// TwinCAT 3 PLC project XtsTransport
// Title: XTS Transport
// Author: D.Hauer
// ProjectVersion: 0.0.1
// Description: basic functionblocks for building XTS transport
// ProgramVersion: 3.1.4026.14
// libraries:
//   Tc2_Math, * (Beckhoff Automation GmbH)
//   Tc2_MC2, * (Beckhoff Automation GmbH)
//   Tc2_Standard, * (Beckhoff Automation GmbH)
//   Tc2_System, * (Beckhoff Automation GmbH)
//   Tc2_Utilities, * (Beckhoff Automation GmbH)
//   Tc3_McCollisionAvoidance, * (Beckhoff Automation GmbH)
//   Tc3_McCoordinatedMotion, * (Beckhoff Automation GmbH)
//   Tc3_Module, * (Beckhoff Automation GmbH)
//   Tc3_XTS_Utility, * (Beckhoff Automation GmbH)
//   VisuDialogs, * (System)
// project tree:
//   APPLICATION/ MAIN_APP.TcPOU, fb_Application.TcPOU, GVL_APPLICATION.TcGVL, PROCESS_HANDSHAKE.TcPOU
//   APPLICATION/Process_Instances/ fb_BufferInfeed.TcPOU, fb_BufferOutfeedRobot.TcPOU, fb_Infeed.TcPOU, fb_OutfeedRobot.TcPOU, fb_SenderBufferInfeed.TcPOU, fb_SenderFast.TcPOU
//   APPLICATION/_types/Application/ E_APP_CHECK.TcDUT (not stored), ST_APP_CTRL.TcDUT (not stored), ST_APP_STATE.TcDUT
//   APPLICATION/_types/Collector/ E_PROCESS_CHECK.TcDUT, E_PROCESS_CTRL.TcDUT, E_PROCESS_STATE.TcDUT (not stored), fb_ProcessCollector.TcPOU, fb_StationCollector.TcPOU, I_ProcessCollector.TcIO, ST_PROCESS_CTRL.TcDUT, ST_PROCESS_STATE.TcDUT, T_PROCESS.TcDUT
//   APPLICATION/_types/Instance/ E_INSTANCE.TcDUT, E_INSTANCE_CHECK.TcDUT (not stored), E_INSTANCE_CMD.TcDUT, E_INSTANCE_STATE.TcDUT, fb_Instance.TcPOU, ST_INSTANCE_CTRL.TcDUT (not stored), ST_INSTANCE_STATE.TcDUT
//   APPLICATION/_types/LinkedList/ fb_Process_LinkedListCtrl.TcPOU, I_Process_LinkedList.TcIO (not stored), ST_PROCESS_DATA.TcDUT, ST_PROCESS_LIST_RESULT.TcDUT (not stored)
//   APPLICATION/_Visu/ SIM_TEST.TcVIS
//   APPLICATION/_Visu/textlists/ TL_E_INSTANCE.TcTLO, TL_E_INSTANCE_CMD.TcTLO (not stored)
//   / GlobalTextList.TcGTLO, MAIN.TcPOU, PLC_1.TcTTO (not stored)
//   MSG/ fb_LocalTime.TcPOU (not stored), f_MessageSet.TcPOU (not stored), GVL_MSG.TcGVL (not stored), MessageData.TcPOU, T_MESSAGE_LIST.TcVIS
//   MSG/types/ e_Device.TcDUT (not stored), E_MessageType.TcDUT (not stored), E_MESSAGE_STATE.TcDUT, e_Subdevice.TcDUT, ST_Message.TcDUT (not stored), TL_E_MESSAGETYPE.TcTLO (not stored)
//   UML/ CD_APPLICATION.TcCD (not stored), CD_GroupCa.TcCD (not stored)
//   XTS/CaGroup/ FB_CaGroup.TcPOU, I_XtsTransport_CaGroup.TcIO
//   XTS/CaGroup/types/ E_CA_GROUP_STATE.TcDUT (not stored), E_GROUP_CHECK.TcDUT (not stored), ST_GROUP_INFO.TcDUT (not stored)
//   XTS/ GVL_XTS.TcGVL, XTS_Parameter.TcGVL
//   XTS/Mover/ fb_Mover.TcPOU, fb_MoverCtrl.TcPOU (not stored), I_XtsTransport_Mover.TcIO
//   XTS/Mover/types/ E_MOVER_CTRL.TcDUT (not stored), E_MOVER_STATE.TcDUT (not stored), ST_GEAR_DATA.TcDUT (not stored), ST_MOVER_CTRL.TcDUT (not stored), ST_MOVER_INFO.TcDUT (not stored), ST_MOVER_STATE.TcDUT (not stored), ST_MOVE_DATA.TcDUT (not stored)
//   XTS/XtsStation/ fb_Station.TcPOU, I_XtsTransport_Station.TcIO
//   XTS/XtsStation/_types/ E_STATION_CTRL.TcDUT, E_STATION_STATE.TcDUT (not stored), fb_Station_LinkedListCtrl.TcPOU, I_Station_LinkedList.TcIO (not stored), ST_STATION_CTRL.TcDUT (not stored), ST_STATION_LIST_RESULT.TcDUT (not stored), ST_STATION_MOVER_DATA.TcDUT (not stored), ST_STATION_PARAMETER.TcDUT (not stored), ST_STATION_STATE.TcDUT, T_NEST_OFFSET.TcDUT (not stored)
//   XTS/_Visualization/ GROUP_VISU.TcVIS, MOVER_VISU.TcVIS, STATION_VISU.TcVIS, Visualization Manager.TcVMO (not stored), XTS_TRANSPORT.TcVIS, XPU_VISU.TcVIS
//   XTS/_Visualization/textlists/ TL_E_CTRL_MOVER.TcTLO (not stored), TL_E_CTRL_STATION.TcTLO (not stored), TL_E_CTRL_TRANSPORT.TcTLO, TL_E_CTRL_XPU.TcTLO
//   XTS/Xpu/ fb_Xpu.TcPOU, fb_XpuCtrl.TcPOU (not stored)
//   XTS/Xpu/types/ E_XPU_CHECK.TcDUT (not stored), E_XPU_CTRL.TcDUT (not stored), E_XPU_INIT.TcDUT, E_XPU_STATE.TcDUT (not stored), ST_XPU_CTRL.TcDUT (not stored), ST_XPU_INFO.TcDUT (not stored), ST_XPU_STATE.TcDUT (not stored)
//   XTS/XtsTransportUnit/ fb_TransportUnit.TcPOU
//   XTS/XtsTransportUnit/types/ E_XTS_TRANSPORT_CHECK.TcDUT (not stored), E_XTS_TRANSPORT_CTRL.TcDUT, E_XTS_TRANSPORT_STATE.TcDUT, ST_XTS_TRANSPORT_CTRL.TcDUT (not stored), ST_XTS_TRANSPORT_STATE.TcDUT (not stored)
//   XTS/_types/ E_PROGRESS.TcDUT (not stored), f_GetProgress.TcPOU (not stored), f_GetState.TcPOU (not stored)

// ---- APPLICATION/_types/Application/ST_APP_STATE.TcDUT
TYPE ST_APP_STATE :
STRUCT
  AppState            : E_INSTANCE_STATE;
  InstanceStates      : REFERENCE TO ARRAY[1..MAX_PROCESS] OF ST_INSTANCE_STATE;
  XtsTransportState   : REFERENCE TO ST_XTS_TRANSPORT_STATE;
END_STRUCT
END_TYPE

// ---- APPLICATION/_types/Collector/E_PROCESS_CHECK.TcDUT
{attribute 'strict'}
{attribute 'to_string'}
TYPE E_PROCESS_CHECK :
(
  PROCESS_CHECK_NULL,
  PROCESS_CHECK_CTRL_REFERENCE_INVALID,
  PROCESS_CHECK_STATE_REFERENCE_INVALID,
  PROCESS_CHECK_MOVER_INFO_REFERENCE_INVALID,
	PROCESS_CHECK_STATION_FIRST_ZERO,
  PROCESS_CHECK_STATION_LAST_ZERO,
  PROCESS_CHECK_STATION_FIRST_MAX,
  PROCESS_CHECK_STATION_LAST_MAX,
  PROCESS_CHECK_STATION_COUNT_NEGATIVE, // last station must have higher index than first station, range must also be closed
  PROCESS_CHECK_STATION_COUNT_TOO_HIGH, // process can only be max (SIZEOF(T_PROCESS)*8)


  PROCESS_CHECK_DONE    := 10000
);
END_TYPE

// ---- APPLICATION/_types/Collector/E_PROCESS_CTRL.TcDUT
{attribute 'qualified_only'}
{attribute 'strict'}
{attribute 'to_string'}
TYPE E_PROCESS_CTRL :
(
  PROCESS_INIT              := 10,
  PROCESS_DISABLE           := 20,
  PROCESS_ENABLE            := 30,
  PROCESS_STATIONS_INFEED,

  PROCESS_STATIONS_ENTER    := 40,
  PROCESS_STATIONS_SEND,

  PROCESS_START             := 60,
  PROCESS_DONE              := 70,
  PROCESS_STATIONS_OUTFEED  := 80
);
END_TYPE

// ---- APPLICATION/_types/Collector/ST_PROCESS_CTRL.TcDUT
TYPE ST_PROCESS_CTRL :
STRUCT
  Cmd               : E_PROCESS_CTRL;
  ProcessTarget     : UINT;
  ActivateStation   : T_PROCESS;  // every bit is a XtsStation
  NestMask          : BYTE;       // every bit is a PosStop in a XtsStation, one mask for all XtsStations, copied to every XtsStation control in process
END_STRUCT
END_TYPE

// ---- APPLICATION/_types/Collector/ST_PROCESS_STATE.TcDUT
TYPE ST_PROCESS_STATE :
STRUCT
  State           : E_PROCESS_STATE;
  Result          : E_PROGRESS;
  Check           : E_PROCESS_CHECK;
END_STRUCT
END_TYPE

// ---- APPLICATION/_types/Collector/T_PROCESS.TcDUT
TYPE T_PROCESS : DWORD; END_TYPE

// ---- APPLICATION/_types/Instance/E_INSTANCE.TcDUT
{attribute 'qualified_only'}
//{attribute 'strict'}
{attribute 'to_string'}
TYPE E_INSTANCE :
(
  // process identifiers as enum, 
  // this enum must not have gaps!
  INVALID,
  BUFFER_INFEED,        // process for getting the job from transfersystem
  INFEED,               // process for getting workpieces from transfersystem
  //OUTFEED_CLAMP,        // process for unloading (12 movers with possible gaps)
  BUFFER_OUTFEED_ROBOT, // process for dealing movers into robot outfeed with no gaps
  OUTFEED_ROBOT_R1,     // process for robot outfeed (12 movers)
  OUTFEED_ROBOT_R2,     // process for robot outfeed (12 movers)
  //SENDER_SLOW,          // process for slowing down movers
  SENDER_FAST,          // process for accelerating movers to return with max velo
  SENDER_BUFFER_INFEED, // process for dealing movers into BUFFER_INFEED, since the curve is vertical, there has to be room when movers are set in motion
  INSTANCE_MAX
)UINT;
END_TYPE

// ---- APPLICATION/_types/Instance/E_INSTANCE_CMD.TcDUT
{attribute 'qualified_only'}
{attribute 'strict'}
{attribute 'to_string'}
TYPE E_INSTANCE_CMD : // instructions for fb_Instance executions
(
	NULL,
  INIT,
  DISABLE,
  ENABLE,
  WORK,
  PROCEED := 100,
  FINISH,
  CLEAR
)UINT;
END_TYPE

// ---- APPLICATION/_types/Instance/E_INSTANCE_STATE.TcDUT
{attribute 'qualified_only'}
//{attribute 'strict'}
{attribute 'to_string'}
TYPE E_INSTANCE_STATE :
(
  NULL,
	INVALID,
  INIT,
  DISABLED,
  DETECT_IN_LIST,
  ENABLED,
  WORKING,
  PROCEEDING,
  FINISH,
  CLEARED
)UINT;
END_TYPE

// ---- APPLICATION/_types/Instance/ST_INSTANCE_STATE.TcDUT
TYPE ST_INSTANCE_STATE :
STRUCT
  State     : E_INSTANCE_STATE;
  Progress  : E_PROGRESS;
END_STRUCT
END_TYPE

// ---- APPLICATION/_types/LinkedList/ST_PROCESS_DATA.TcDUT
TYPE ST_PROCESS_DATA :
STRUCT
  {attribute 'displaymode':='bin'}
  wTarget             : T_PROCESS; // where and how many stations are to be used in process
END_STRUCT
END_TYPE

// ---- MSG/types/E_MESSAGE_STATE.TcDUT
{attribute 'strict'}
TYPE E_MESSAGE_STATE :
(
  MSG_INVALID_POINTERS  := -1,
	MSG_NULL,
  MSG_INIT,
  MSG_ROOT              := 10,
  MSG_ROOT_CREATE,
  MSG_ROOT_CREATE_BUSY,
  MSG_FOLDER,
  MSG_FOLDER_CREATE,
  MSG_FOLDER_CREATE_BUSY,
  MSG_FILE_CREATE_DONE,
  MSG_LINE_START        := 100,
  MSG_LINE_BUILD,
  MSG_LINE_CHECK,
  MSG_WRITE_FILE_BUSY  := 200,
  MSG_WRITE_FILE_END,
  MSG_WRITE_FILE_DONE   := 1000
)DINT;
END_TYPE

// ---- MSG/types/e_Subdevice.TcDUT
{attribute 'strict'}
{attribute 'to_string'}
TYPE e_Subdevice :
(
  // sub device for message system
  General                 :=  0,
  // Motion Control FB Instances
  fbPower,
  fbReset,
  fbResetSercos,
  fbHalt,
  fbStop,                 // 5
  fbHome,
  fbJog,
  fbMoveVelocity1,
  fbMoveVelocity2,
  fbMoveAbsolute1,        // 10
  fbMoveAbsolute2,
  fbMoveEndless,
  fbMovePtP,
  fbMoveVelo,

  // CA CollisionAvoidance FB instances
  // CA group fb instances
  fbCaGroup             := 30,
  fbMoveToPosCa,
  fbSendToAbsPosCa,
  fbSendToModuloPosCa,
  fbGearInPosCa,
  fbGroupAddAxis,
  fbGroupRemoveAxis,
  fbGroupDisable,
  fbGroupEnable,
  fbGroupErrorRead,
  fbGroupStatusRead,
  fbGroupReset,
  fbGroupStop,
  fbHaltCa,

  fbGearIn                := 50,
  fbGearOut,
  fbGearInMultiMaster,

  fbCamOutV2              := 80,
  fbCamInV2,
  fbCamScalingV2,
  fbCamInfoV2,
  fbReadMotionFunction,
  fbReadMotionFunctionPoint,
  fbReadMotionFunctionValues,
  fbWriteMotionFunction,
  fbWriteMotionFunctionPoint,
  fbSetOnlineChangeMode,

  fbReadParameter         := 100,
  fbReadBoolParameter,
  fbWriteParameter,
  fbWriteBoolParameter,
  fbWriteParameterPersistent,

  fbBuildGroup            := 200,
  fbClearGroup,
  fbLoadProg,
  fbResetItp,
  fbStartStopItp,
  fbEStopItp,             // 205
  fbStepOnAfterEStopItp,
  fbConfirmHskItp,
  fbDelDtgItp,
  fbNciFeedTablePreparation,
  fbNciFeedTable,         // 210
  fbReadLine,
  fbItpReadRParams,
  fbItpWriteRParams,
  Get_ItpState,
  Get_Error,              // 215


  XfcPositionAtTime       := 300,
  XfcTimeOfPosition,
  XfcTimeToPosition,
  XfcTimeToModuloPosition,
  XfcRecordedPosition,
  XfcTouchProbe,          // 305
  XfcTouchProbeEL1258,
  XfcTouchProbeOptions,
  XfcTriggerRef,
  XfcTriggerRef_MT,
  XfcEl1258Interface_MT,  // 310
  XfcRecordedPosition_MT,
  XfcTriggerOut,
  XfcTriggerStart,
  XfcSwitchOn_2252,
  XfcSwitchOff_2252,      // 315
  XfcInit,
  XfcLatchPosition,
  XfcWaitForPosition,

  AxisMode              := 1000,
  AxisControl,

  NciControl            := 2000,
  NciStartUp,
  NciCycle,
  NciIdle,

  StationLinkedList     := 3000,
  StationInitList,
  StationAddHead,
  StationAddTail,
  StationGetHead,
  StationRemoveHeadValue,

  StationControl        := 4000,
  StationState, 

  Xpu_fbEnvironment     := 5000,
  Xpu_fbProcessingUnit,
  Xpu_fbXpuPart,
  Xpu_fbXpuTrack,
  Xpu_fbMc2CaGroup,
  Xpu_fbParameterSet,

  Xpu_fbPartModules     := 5500,

  Xpu_fbMoverXpu        := 6000,

  TransportUnit_General := 7000,
  TransportUnit_Restart := 7010,
  TransportUnit_Start,
  TransportUnit_XpuInit,

  CamControl            := 8000,
  CamStartUp,
  CamCycle,

  Process_StationCollector    := 11000,
  Process_ProcessCollector    := 11100,
  Process_ProcessCollector_Init,
  Process_ProcessCollector_Cycle,
  Process_ProcessCollector_Control,

  Process_LinkedList_GetHead,
  Process_LinkedList_RemoveHead,
  Process_LinkedList_AddTail,
  Process_LinkedList_CheckData,

  Instance_BufferInfeed       := 12000,
  Instance_BufferInfeed_CheckDisabled,
  Instance_BufferInfeed_CheckEnabled,
  Instance_BufferInfeed_CheckInfeed,
  Instance_BufferInfeed_CheckOutfeed,
  Instance_BufferInfeed_CheckTarget,
  Instance_Infeed,
  Instance_BufferOutfeedRobot,
  Instance_OutfeedRobot_R1,
  Instance_OutfeedRobot_R2,
  Instance_Sender_Fast,
  Instance_Sender_BufferInfeed,

  Application                 := 13000,
  Application_Check,
  Application_Clear,
  Application_Cmd,
  Application_Disable,
  Application_Enable,
  Application_Finish,
  Application_Init,
  Application_Proceed,
  Application_Work

)DINT;
END_TYPE

// ---- XTS/XtsStation/_types/E_STATION_CTRL.TcDUT
{attribute 'qualified_only'}
{attribute 'strict'}
{attribute 'to_string'}
TYPE E_STATION_CTRL :
(
  STATION_CTRL_NULL,              // nothing happens here
	STATION_INIT            := 1,   // hard reset of station, list is cleared
  STATION_DISABLE         := 10,  // 
  STATION_ENABLE,                 // 

  STATION_MOVER_ENTER     := 20,  // mover may enter station
  STATION_MOVER_ENTER_RETRY,      // retry after E_STATION_STATE.STATION_ERROR_INFEED_ERROR
  STATION_MOVER_SEND,             // do not enter, send to E_STATION_STATE.STATION_MOVER_OUT

  STATION_PROCESS_START   := 30,  // double handshake with extern
  STATION_PROCESS_DONE,           // single handshake with extern

  STATION_MOVER_OUT       := 50,  // mover may leave station now; ticket for mover is checked here (ST_STATION_CTRL.nTargetStation)
  STATION_MOVER_OUT_RETRY,        // retry after E_STATION_STATE.STATION_ERROR_OUTFEED_ERROR

  STATION_MOVER_GONE      := 60   // mover has left station, last handshake station is empty

)USINT;
END_TYPE

// ---- XTS/XtsStation/_types/ST_STATION_STATE.TcDUT
{attribute 'pack_mode' := '2'}
TYPE ST_STATION_STATE :
STRUCT
  eState          : E_STATION_STATE;
  {attribute 'displaymode':='bin'}
  nMask           : BYTE;
  nMoverId        : USINT;
  rMoverModPos    : LREAL; // modulo position of detected mover
  rMoverVelo      : LREAL;
  rMoverAcc       : LREAL;
  nQueue          : USINT; // queue count for station
END_STRUCT
END_TYPE

// ---- XTS/Xpu/types/E_XPU_INIT.TcDUT
{attribute 'to_string'}
TYPE E_XPU_INIT :
(
	INIT_START,
  INIT_ENVIRONMENT_OID            := 10,
  INIT_INFO_SERVER_ITF,
  INIT_INFO_SERVER_STATION_COUNT,
  INIT_INFO_SERVER_STATION_OID,
  INIT_CA_GROUP_OID               := 20,
  INIT_CA_GROUP_GET_OID,
  INIT_CA_GROUP_CHECK_OID,
  INIT_CA_GROUP_COM,
  INIT_PARAMETERSET_COUNT,
  INIT_PARAMETERSET_OID,
  INIT_PARAMETERSET_COM,
  INIT_PARAMETERSET_COM_NEXT,
  INIT_PROCESSING_UNIT_COM        := 30,
  INIT_PROCESSING_UNIT_PART_COUNT,
  INIT_PROCESSING_UNIT_PART_OID,
  INIT_PROCESSING_UNIT_TRACK_COUNT,
  INIT_PROCESSING_UNIT_TRACK_OID,
  INIT_PROCESSING_UNIT_MOVER_COUNT,
  INIT_PROCESSING_UNIT_MOVER_OID,
  INIT_PROCESSING_UNIT_TASK_COUNT,
  INIT_PROCESSING_UNIT_TASK_OID,
  INIT_TRACK_COM                  := 50,
  INIT_PART_COM                   := 60,
  INIT_PART_MODULE_COUNT,
  INIT_PART_MODULE_OID,
  INIT_PART_MODULE_COM,
  INIT_PART_MODULE_COM_NEXT,
  INIT_MOVER_COM                  := 70,
  INIT_MOVER_COM_NEXT,
  INIT_DATA_GET                   := 90,
  INIT_DATA_CHECK,
  INIT_DONE                       := 100
)UINT;
END_TYPE

// ---- XTS/XtsTransportUnit/types/E_XTS_TRANSPORT_CTRL.TcDUT
{attribute 'strict'}
{attribute 'to_string'}
TYPE E_XTS_TRANSPORT_CTRL :
(
  CMD_NULL,
  CMD_INIT                  := 10,  // Xpu, Group, Mover initialization: clear errors, clear group, check Xpu data, check mover detection
  CMD_IDLE,

  CMD_MOVER_ENABLE          := 20,  // all mover are enabled, checked for ControlLoopClosed
  CMD_MOVER_DISABLE,                // all mover are disabled, no axis in CaGroup: no error, any axis in CaGroup: group error
  CMD_MOVER_HALT_CA,                // all movers are stopped with MC_HaltCA[]. ONLY use if all movers are in CA group

  CMD_GROUP_CLEAR           := 30,  // halt all movers, clear errors, remove all movers from group, clear group
  CMD_GROUP_BUILD,                  // add all movers to group
  CMD_GROUP_ENABLE,                 // group with movers is enabled
  CMD_GROUP_STOP,                   // moving CA Group is stopped

  CMD_TRANSPORT_START       := 40,  // move all mover[i] to start position
  CMD_TRANSPORT_RESTART             // move all mover[i] to LastPosition[i]

)UINT;
END_TYPE

// ---- XTS/XtsTransportUnit/types/E_XTS_TRANSPORT_STATE.TcDUT
{attribute 'to_string'}
TYPE E_XTS_TRANSPORT_STATE :
(
  TRANSPORT_NULL,
  TRANSPORT_INVALID,
  TRANSPORT_INIT            := 10,  // Xpu, Group, Mover initialization: init TcCOM objects, clear errors, clear group, check Xpu data, check mover detection
  TRANSPORT_IDLE,                   // cyclic check for errors, check Xpu data

  TRANSPORT_MOVER_ENABLE    := 20,  // all mover are enabled, checked for ControlLoopClosed
  TRANSPORT_MOVER_DISABLE,          // all mover are disabled
  TRANSPORT_MOVER_HALT_CA,          // all mover standstill
  TRANSPORT_MOVER_STOP,

  TRANSPORT_GROUP_CLEAR     := 30,  // halt all movers, clear errors, remove all movers from group, clear group
  TRANSPORT_GROUP_BUILD,            // add all movers to group
  TRANSPORT_GROUP_ENABLE,           // group with movers is enabled
  TRANSPORT_GROUP_STOP,             // CaGroup Stop, CaGroup Reset, All movers halt

  TRANSPORT_START           := 40,  // move all mover[i] to start position
  TRANSPORT_RESTART                 // move all mover[i] to LastPosition[i]
)UINT;
END_TYPE

// ---- APPLICATION/GVL_APPLICATION.TcGVL
VAR_GLOBAL CONSTANT
  MAX_PROCESS         : E_INSTANCE := E_INSTANCE.SENDER_BUFFER_INFEED;
END_VAR
{attribute 'qualified_only'}
VAR_GLOBAL
  //-----------------------------------------------------------------------------------------------
  // Application
  //
  //  this is the part you will have to change and adapt into your programming
  //-----------------------------------------------------------------------------------------------
  //-----------------------------------------------------------------------------------------------
  // fb_Application:
  // - procedures for getting fb_Instance classes and XTS_TRANSPORT_LAYER to work
  //
  //  - Cmd/state behaviour as in fb_TransportUnit
  //  - E_INSTANCE_CMD  / E_INSTANCE_STATE + E_PROGRESS
  //      INIT          /   INIT          : initialize processes and XtsStations       
  //      DISABLE       /   DISABLED      : RemoveAllAxis from CA Group, disable CA Group, disable all movers
  //      ENABLE        /   ENABLED       : AddAllAxis to CA Group, Enable CA Group, Enable all movers
  //      WORK          /   WORKING       : CMD_TRANSPORT_START, enable handshakes, start writing list entries to BUFFER_INFEED
  //      PROCEED       /   PROCEEDING    : CMD_TRANSPORT_RESTART, enable handshakes, continue writing list entries to BUFFER_INFEED
  //      FINISH        /   FINISH        : stop writing list entries to BUFFER_INFEED, handshake processes until outfeeds are empty
  //      CLEAR         /   CLEARED       : clear all instances of fb_Instance, clear all XtsStations
  //-----------------------------------------------------------------------------------------------
  ApplicationMain       : fb_Application;
  AppControl            : ST_APP_CTRL;
  AppState              : ST_APP_STATE;


  //-----------------------------------------------------------------------------------------------
  // Process instances
  //  - processes are similar but also different, hence working with inheritance of fb_Instance
  //  - change/check here if you need a process procedure that matches your use case
  //-----------------------------------------------------------------------------------------------
  BufferInfeed          : fb_BufferInfeed;        // prepare movers to enter infeed station
  Infeed                : fb_Infeed;              // infeed into XTS, transfersystem drops its load here
  BufferOutfeedRobot    : fb_BufferOutfeedRobot;  // feeds 24 Mover into 2 processes (12 each), no gaps
  Outfeed_R1            : fb_OutfeedRobot;        // unloads 12 mover
  Outfeed_R2            : fb_OutfeedRobot;        // unloads 12 mover
  SenderFast            : fb_SenderFast;          // every passing mover is accelersted to max velo
  SenderBufferInfeed    : fb_SenderBufferInfeed;  // checks if there is room for 12-x mover, sends mover to BufferInfeed for a new round


  //-----------------------------------------------------------------------------------------------
  // fb_Instance control and state
  //  - structs are used in fb_Application as reference 
  //-----------------------------------------------------------------------------------------------
  InstanceCtrl          : ARRAY[1..MAX_PROCESS] OF ST_INSTANCE_CTRL;
  InstanceState         : ARRAY[1..MAX_PROCESS] OF ST_INSTANCE_STATE;


  //-----------------------------------------------------------------------------------------------
  // Linked List instances
  //  - THIS example only uses the linked list in fb_BufferInfeed 
  //    as buffered input from an extern transfersystem
  //-----------------------------------------------------------------------------------------------
  ProcessList           : ARRAY[1..MAX_PROCESS] OF fb_Process_LinkedListCtrl; // information transfer between processes
  ItfProcessList        : ARRAY[1..MAX_PROCESS] OF I_Process_LinkedList;      // use this interface in your function blocks


  //-----------------------------------------------------------------------------------------------
  // Collector instances
  //
  //  - layer for grouping parallel XtsStations for process handshakes
  //-----------------------------------------------------------------------------------------------
  //  - fb_ProcessCollector:
  //    - uses .ProcessCtrl and .ProcessState for handshakes with application
  //
  //    - .ActivateStation is evaluated after enabling infeed in state 
  //      E_PROCESS_STATE.PROCESS_DISABLE:/E_PROGRESS.PROGRESS_BUSY:
  //      
  //    - ST_PROCESS_STATE:
  //      - contains 3 enumerations for you to check
  //      - State           : E_PROCESS_STATE;
  //        - main state for handshakes
  //
  //      - Result          : E_PROGRESS;
  //        - substate for checks during handshake; 
  //          PROGRESS_BUSY --> handshakes are accepted (see fb_ProcessCollecotr.Cycle())
  //
  //      - Check           : E_PROCESS_CHECK;
  //        - cyclic pointer check: use this on startup of your application
  //
  //    - inherits fb_StationCollector
  //-----------------------------------------------------------------------------------------------
  ProcessCollector      : ARRAY[1..MAX_PROCESS] OF fb_ProcessCollector;       // grouping of XtsStations
  ItfProcessCollector   : ARRAY[1..MAX_PROCESS] OF I_ProcessCollector;        // interface for use in your function blocks like BufferInfeed etc.
END_VAR

// ---- XTS/GVL_XTS.TcGVL
{attribute 'qualified_only'}
VAR_GLOBAL
  //---------------------------------------------------------------------------
  // XTS Station
  //  - handshakes mover in station with extern control
  //  - station parameters (positions, gap, dyn. constraints, description...)
  StationStart        : ST_STATION_PARAMETER;   // Xts transport is sending all mover to this position (CMD_TRANSPORT_START)
  StationStartIndex   : UINT := 52;             // index of XtsStation where all movers are entered into linked list.

  // station handshaking with mover and extern process
  // station sends mover to target station/WaitPos
  // station adds mover data to LinkedList.AddTail() of target station
  Station             : ARRAY[1..MAX_STATION] OF fb_Station;
  StationList         : ARRAY[1..MAX_STATION] OF fb_Station_LinkedListCtrl;

  StationQueue        : ARRAY[1..MAX_STATION]    OF 
                        ARRAY[1..MAX_LIST_NODES] OF ST_STATION_MOVER_DATA;

  // interface for access to List methods
  StationListItf      : ARRAY[1..MAX_STATION] OF I_Station_LinkedList;

  // interface for access to station methods
  StationCtrlItf      : ARRAY[1..MAX_STATION] OF I_XtsTransport_Station;

  // ctrl / state datafields for extern control
  StationCtrl         : ARRAY[1..MAX_STATION] OF ST_STATION_CTRL;   // control for extern to write
  StationState        : ARRAY[1..MAX_STATION] OF ST_STATION_STATE;  // state for extern to read

  // station parameter
  StationParameter    : ARRAY[1..MAX_STATION] OF ST_STATION_PARAMETER;

  // static position offsets in stations
  PositionOffset      : ARRAY[1..MAX_STATION] OF T_NEST_OFFSET;


  //---------------------------------------------------------------------------
  // XTS
  // XTS TransportUnit
  //  - handles request for XPU, Group, Mover, StartUp, ReStart
  XtsTransport        : fb_TransportUnit;         // manages members of XTS transport for extern to access

  XtsTransportCtrl    : ST_XTS_TRANSPORT_CTRL;    // control of XTS transport for extern to write
  XtsTransportState   : ST_XTS_TRANSPORT_STATE;   // state   of XTS transport for extern to read


  //---------------------------------------------------------------------------
  // XPU
  // XTS-Utility checks
  Xpu             : fb_XpuCtrl;

  XpuCtrl         : ST_XPU_CTRL;
  XpuState        : ST_XPU_STATE;
  XpuInfo         : ST_XPU_INFO;
  XpuModules      : ARRAY[1..MAX_MODULE] OF Tc3_XTS_Utility.ST_InfoDataView;


  //---------------------------------------------------------------------------
  // Collision avoidance group CA
  //
  // - add mover to group
  // - build group
  // - clear group
  CaGroup         : FB_CaGroup;                   // cyclic check of CaGroup state and errors; carries methods for handling CaGroup
  CaGroupItf      : I_XtsTransport_CaGroup;       // Interface used by fb_TransportUnit

  // cyclic mapping to MOTION/Objects/CaGroup 
  CaGroupRef      : Tc3_McCoordinatedMotion.AXES_GROUP_REF;

  // Info data from CaGroup FB
  CaGroupInfo     : ST_GROUP_INFO;                // cyclic info about CaGroup for fb_TransportUnit to read
  //---------------------------------------------------------------------------

  //---------------------------------------------------------------------------
  // MC2 encapsulation, CA movement
  Mover           : ARRAY[1..MAX_MOVER] OF fb_MoverCtrl;    // MC and CA methods for mover; cyclic check for individual command on mover

  MoverCtrl       : ARRAY[1..MAX_MOVER] OF ST_MOVER_CTRL;   // control of individual mover for extern to write
  MoverState      : ARRAY[1..MAX_MOVER] OF ST_MOVER_STATE;  // state   of individual mover for extern to read

  MoverItf        : ARRAY[1..MAX_MOVER] OF I_XtsTransport_Mover;  // Interface used by fb_TransportUnit

  LastPosition    : ARRAY[1..MAX_MOVER] OF LREAL;           // on execute of any movement, value is saved here (used by fb_Mover)
  LastGap         : ARRAY[1..MAX_MOVER] OF LREAL;           // on execute of any movement, value is saved here (used by fb_Mover)

  MoverInfo       : ARRAY[1..MAX_MOVER] OF ST_MOVER_INFO;   // cyclic info about mover for extern to read

  MoveData        : ARRAY[1..MAX_MOVER] OF ST_MOVE_DATA;    // dynamic constraints for move commands
  GearData        : ARRAY[1..MAX_MOVER] OF ST_GEAR_DATA;    // dynamic constraints and positions for GearIn/GearInPosCa
  
  // cyclic mapping to MOTION/Axes
  AxisRefMover    : ARRAY[1..MAX_MOVER] OF Tc2_MC2.AXIS_REF;
  //---------------------------------------------------------------------------
END_VAR

// ---- XTS/XTS_Parameter.TcGVL
//{attribute 'qualified_only'}
VAR_GLOBAL CONSTANT
// HAUD 2025 06 04
//
//    XTS_TRANSPORT_LAYER project
//    
//    MIT License
//    
//    Copyright (c) 2025 HAUD
//    
//    Permission is hereby granted, free of charge, to any person obtaining a copy
//    of this software and associated documentation files (the "Software"), to deal
//    in the Software without restriction, including without limitation the rights
//    to use, copy, modify, merge, publish, distribute, sublicense, and/or sell
//    copies of the Software, and to permit persons to whom the Software is
//    furnished to do so, subject to the following conditions:
//    
//    The above copyright notice and this permission notice shall be included in all
//    copies or substantial portions of the Software.
//    
//    THE SOFTWARE IS PROVIDED "AS IS", WITHOUT WARRANTY OF ANY KIND, EXPRESS OR
//    IMPLIED, INCLUDING BUT NOT LIMITED TO THE WARRANTIES OF MERCHANTABILITY,
//    FITNESS FOR A PARTICULAR PURPOSE AND NONINFRINGEMENT. IN NO EVENT SHALL THE
//    AUTHORS OR COPYRIGHT HOLDERS BE LIABLE FOR ANY CLAIM, DAMAGES OR OTHER
//    LIABILITY, WHETHER IN AN ACTION OF CONTRACT, TORT OR OTHERWISE, ARISING FROM,
//    OUT OF OR IN CONNECTION WITH THE SOFTWARE OR THE USE OR OTHER DEALINGS IN THE
//    SOFTWARE.

  Version             : STRING  := '4.00.08';

  MAX_MOVER           : UINT    := TO_UINT(Tc3_XTS_Utility.TcIoXtsEnvironmentParameterList.MaxXtsMoversPerXpu);
  MAX_MODULE          : UINT    := TO_UINT(Tc3_XTS_Utility.TcIoXtsEnvironmentParameterList.MaxModulesPerPart);
  MAX_PART            : UINT    := TO_UINT(Tc3_XTS_Utility.TcIoXtsEnvironmentParameterList.MaxXtsPartsPerXpu);
  MAX_TRACK           : UINT    := TO_UINT(Tc3_XTS_Utility.TcIoXtsEnvironmentParameterList.MaxXtsTracksPerXpu);
  MAX_GROUP           : UINT    := TO_UINT(Tc3_XTS_Utility.TcIoXtsEnvironmentParameterList.MaxXtsCaGroup);

  MAX_INFO_SERVER     : UINT    := TO_UINT(Tc3_XTS_Utility.TcIoXtsEnvironmentParameterList.MaxXtsInfoServer);
  MAX_INFO_STATION    : UINT    := TO_UINT(Tc3_XTS_Utility.TcIoXtsEnvironmentParameterList.MaxXtsInfoStation);
  MAX_INFO_STOP_POS   : UINT    := TO_UINT(Tc3_XTS_Utility.TcIoXtsEnvironmentParameterList.MaxXtsStopPositionsPerStation);

  MAX_PARAMETER_SET   : UINT    := TO_UINT(Tc3_XTS_Utility.TcIoXtsEnvironmentParameterList.MaxXtsParameterSet);

  MAX_NCT_BASE_UNIT   : UINT    := TO_UINT(Tc3_XTS_Utility.TcIoXtsEnvironmentParameterList.MaxXtsNctBaseUnitInterfaces);

  MAX_STATION         : UINT    := 53;
  MAX_STATION_NEST    : UINT    := TO_UINT(SIZEOF(ST_STATION_STATE.nMask)*8);
  // MAX_LIST_NODES      : UINT    := MAX_MOVER;
  MAX_LIST_NODES      : UINT    := 108; // visualization can not handle access to MAX_MOVER
  MAX_MASTER          : UINT    := 1;
END_VAR

// ---- APPLICATION/_types/Collector/I_ProcessCollector.TcIO
INTERFACE I_ProcessCollector

PROPERTY ActivateStation : DWORD // bit mask for enabling XtsStations in Process
GET
END_GET
END_PROPERTY

METHOD BitsToString : STRING(SIZEOF(T_PROCESS)*8) // T_PROCESS to string
VAR_INPUT
  inVal       : T_PROCESS;
END_VAR
END_METHOD

METHOD Cycle // cyclic call for checking XtsStation state masks and command input from process
END_METHOD

METHOD PUBLIC DelBit : T_PROCESS
VAR_INPUT
  inVal   : T_PROCESS;
  bitNo   : DINT;
END_VAR
END_METHOD

METHOD PUBLIC GetBit : BOOL
VAR_INPUT
  inVal   : T_PROCESS;
  bitNo   : DINT;
END_VAR
END_METHOD

METHOD GetMoverInStation : ST_MOVER_INFO // mover in station info
VAR_INPUT
  nStation            : UINT;   // index of GVL_XTS.StationState[nStation]
END_VAR
END_METHOD

METHOD GetStationState : ST_STATION_STATE
VAR_INPUT
  nStation            : UINT;   // index of GVL_XTS.StationState[nStation]
END_VAR
END_METHOD

METHOD PUBLIC Init : E_PROGRESS // clears all XtsSubstations, then disables all
VAR_INPUT
  Execute     : BOOL;
END_VAR
END_METHOD

PROPERTY MessageLevel : e_MessageType
GET
END_GET
SET
END_SET
END_PROPERTY

PROPERTY ProcessCtrl : reference to st_process_ctrl
GET
END_GET
SET
END_SET
END_PROPERTY

PROPERTY ProcessId : E_INSTANCE
GET
END_GET
SET
END_SET
END_PROPERTY

PROPERTY ProcessState : reference to st_process_state
GET
END_GET
SET
END_SET
END_PROPERTY

PROPERTY QueueMoverIDs : ARRAY[1..SIZEOF(T_PROCESS)*8] OF UINT
GET
END_GET
END_PROPERTY

PROPERTY QueueProcessCount : UINT // sum of all station queues
GET
END_GET
END_PROPERTY

PROPERTY QueueStationCount : ARRAY[1..SIZEOF(T_PROCESS)*8] OF UINT
GET
END_GET
END_PROPERTY

METHOD PUBLIC SetBit : T_PROCESS
VAR_INPUT
  inVal   : T_PROCESS;
  bitNo   : DINT;
END_VAR
END_METHOD

PROPERTY StationCount : UINT
GET
END_GET
END_PROPERTY

PROPERTY StationFirst : uint
GET
END_GET
SET
END_SET
END_PROPERTY

PROPERTY StationLast : uint
GET
END_GET
SET
END_SET
END_PROPERTY

PROPERTY TargetIndex : ARRAY[1..SIZEOF(T_PROCESS)*8] OF USINT
GET
END_GET
SET
END_SET
END_PROPERTY

PROPERTY TargetMask : ARRAY[1..SIZEOF(T_PROCESS)*8] OF BYTE
GET
END_GET
SET
END_SET
END_PROPERTY

METHOD To_T_Process : T_PROCESS // maps (2^nExp)-1 onto T_PROCESS datatype 
VAR_INPUT
  nExp              : BYTE;
END_VAR
END_METHOD

END_INTERFACE

// ---- XTS/CaGroup/I_XtsTransport_CaGroup.TcIO
INTERFACE I_XtsTransport_CaGroup

METHOD AddAll : E_PROGRESS
VAR_INPUT
  Execute     : BOOL;
END_VAR
END_METHOD

METHOD Disable : E_PROGRESS
VAR_INPUT
  Execute     : BOOL;
END_VAR
END_METHOD

METHOD Enable : E_PROGRESS
VAR_INPUT
  Execute     : BOOL;
END_VAR
END_METHOD

METHOD McHaltAll : E_PROGRESS
VAR_INPUT
  Execute       : BOOL;
END_VAR
END_METHOD

METHOD McResetAll : E_PROGRESS
VAR_INPUT
  Execute       : BOOL;
END_VAR
END_METHOD

METHOD RemoveAll : E_PROGRESS
VAR_INPUT
  Execute     : BOOL;
END_VAR
END_METHOD

METHOD Reset : E_PROGRESS
VAR_INPUT
  Execute     : BOOL;
END_VAR
END_METHOD

METHOD Stop : E_PROGRESS
VAR_INPUT
  Execute     : BOOL;
END_VAR
END_METHOD

END_INTERFACE

// ---- XTS/Mover/I_XtsTransport_Mover.TcIO
INTERFACE I_XtsTransport_Mover

METHOD Disable : E_PROGRESS
VAR_INPUT
  Execute             : BOOL;
END_VAR
END_METHOD

METHOD Enable : E_PROGRESS
VAR_INPUT
  Execute             : BOOL;
END_VAR
END_METHOD

METHOD GearIn : E_PROGRESS;
VAR_INPUT
  Execute             : BOOL;
  stMoveData          : ST_MOVE_DATA;
  stGearData          : ST_GEAR_DATA;
END_VAR
END_METHOD

METHOD GearInPosCa : E_PROGRESS
VAR_INPUT
  Execute             : BOOL;
  stMoveData          : ST_MOVE_DATA;
  stGearData          : ST_GEAR_DATA;  
END_VAR
END_METHOD

METHOD GearOut : E_PROGRESS
VAR_INPUT
  Execute             : BOOL;
END_VAR
END_METHOD

METHOD Halt : E_PROGRESS
VAR_INPUT
  Execute             : BOOL;
  stMoveData          : ST_MOVE_DATA;
END_VAR
END_METHOD

METHOD HaltCa : E_PROGRESS
VAR_INPUT
  Execute             : BOOL;
  stMoveData          : ST_MOVE_DATA;
END_VAR
END_METHOD

PROPERTY MessageLevel : e_messagetype
SET
END_SET
END_PROPERTY

PROPERTY ModuloTurn : dint
GET
END_GET
END_PROPERTY

METHOD MoveToPos : E_PROGRESS
VAR_INPUT
  Execute             : BOOL;
  stMoveData          : ST_MOVE_DATA;
END_VAR
END_METHOD

METHOD MoveToPosCa : E_PROGRESS
VAR_INPUT
  Execute             : BOOL;
  stMoveData          : ST_MOVE_DATA;
END_VAR
END_METHOD

PROPERTY RailLength : LREAL
GET
END_GET
SET
END_SET
END_PROPERTY

METHOD Reset : E_PROGRESS
VAR_INPUT
  Execute             : BOOL;
END_VAR
END_METHOD

METHOD SendToAbsPosCa : E_PROGRESS
VAR_INPUT
  Execute             : BOOL;
  stMoveData          : ST_MOVE_DATA;
END_VAR
END_METHOD

METHOD SendToModuloPosCa : E_PROGRESS
VAR_INPUT
  Execute             : BOOL;
  stMoveData          : ST_MOVE_DATA;
END_VAR
END_METHOD

END_INTERFACE

// ---- XTS/XtsStation/I_XtsTransport_Station.TcIO
INTERFACE I_XtsTransport_Station

METHOD Init : e_progress
VAR_INPUT
END_VAR
END_METHOD

END_INTERFACE

// ---- APPLICATION/fb_Application.TcPOU
//---------------------------------------------------------------------------------------------------------------
//
//  HAUD 2025.03.31
//
//  - EXAMPLE for top level procedures
//    - transport layer
//    - Collector layer
//    - process layer
//    - instance ctrl/state
//
//  - rewrite/change/discard as you require for your application
//
//  - this function block is NOT intended for direct use outside the scope of this example
//  - maybe the command mechanics are useful for your application
//
//---------------------------------------------------------------------------------------------------------------
FUNCTION_BLOCK fb_Application
VAR
  _eCheck                       : E_APP_CHECK;
  _eInit                        : E_PROGRESS;

  _Ctrl                         : REFERENCE TO ST_APP_CTRL;
  _State                        : REFERENCE TO ST_APP_STATE;

  _eResult                      : E_PROGRESS;

  _eCmd,
  _eCmdOld                      : E_INSTANCE_CMD;
  _eState                       : E_INSTANCE_STATE;

  // Transport Ctrl/State
  _XtsTransportCtrl             : REFERENCE TO ST_XTS_TRANSPORT_CTRL;
  _XtsTransportState            : REFERENCE TO ST_XTS_TRANSPORT_STATE;

  _InstanceCtrl                 : REFERENCE TO ARRAY[1..MAX_PROCESS] OF ST_INSTANCE_CTRL;
  _InstanceState                : REFERENCE TO ARRAY[1..MAX_PROCESS] OF ST_INSTANCE_STATE;
  
  _ItfProcessCollector          : REFERENCE TO ARRAY[1..MAX_PROCESS] OF I_ProcessCollector;

  _ItfProcessList               : REFERENCE TO ARRAY[1..MAX_PROCESS] OF I_Process_LinkedList;

  // timers for this example
  _tonProcess                   : ARRAY[1..MAX_PROCESS] OF Tc2_Standard.TON;
  _tProcess                     : ARRAY[1..MAX_PROCESS] OF TIME;


  _stMsg                        : ST_Message;
  _MessageLevel                 : E_MessageType;

  // ListData()
  _nLoadCaseOld,
  _nLoadCase                    : UINT := 0; // 0 = fully loaded, 2 = mod 5 missing 1, 1 = missing up to 11

  // Work()
  _bSingleOutput                : BOOL;

  _nTimeVariantOld,
  _nTimeVariant                 : UINT;

  _sAppState                    : STRING;
  _sAppResult                   : STRING;

  {attribute 'hide'}
  _nAppState                    : E_INSTANCE_STATE;
  {attribute 'hide'}
  _nAppResult                   : E_PROGRESS;
END_VAR

IF NOT Check() THEN RETURN; END_IF
//-----------------------------------------------------------------------------
//-----------------------------------------------------------------------------
// set message device
//-----------------------------------------------------------------------------
_stMsg.eDevice                  := e_Device.Application + 1;

_eCmd                           := _Ctrl.Cmd;
// check for command change
// get state for cmd
IF (_eCmd <> _eCmdOld)
THEN
  _eState                       := Cmd(_eCmd);
  _eCmdOld                      := _eCmd;

  IF (_MessageLevel > E_MessageType.eMessageWarning)
  THEN
    _stMsg.eType                      := E_MessageType.eMessageinfo;
    _stMsg.eSubdevice                 := e_Subdevice.Application_Cmd;
    _stMsg.iErrorNumber               := _eCmd;
    _stMsg.sText                      := concat(TO_STRING(_eCmd), ': ');
    _stMsg.sText                      := concat(_stMsg.sText, TO_STRING(_eState));
    f_MessageSet(_stMsg);
  END_IF
END_IF

CASE _eResult
OF
  E_PROGRESS.PROGRESS_INVALID:
    _State.AppState             := TO_UINT(_eResult);

  E_PROGRESS.PROGRESS_ERROR:
    _State.AppState             := _eState + E_PROGRESS.PROGRESS_ERROR;

  E_PROGRESS.PROGRESS_DONE:
    _State.AppState             := _eState + E_PROGRESS.PROGRESS_DONE;

    IF (_XtsTransportState.GroupInfo.GroupErrorStop) OR
       (_XtsTransportState.GroupInfo.GroupError)     OR
       NOT (_XtsTransportState.XpuInfo.AllPositionsValid)
    THEN
      _eResult                  := E_PROGRESS.PROGRESS_ERROR;
    END_IF
ELSE
  _State.AppState               := _eState + _eResult;

  CASE _eState
  OF
    E_INSTANCE_STATE.INIT:
      _eInit := _eResult        := Init(TRUE);
  
    E_INSTANCE_STATE.DISABLED:
      _eResult                  := Disable(TRUE);
  
    E_INSTANCE_STATE.ENABLED:
      IF NOT (_XtsTransportState.XpuState.DcLink) OR
         NOT (_XtsTransportState.XpuInfo.AllPositionsValid)
      THEN
        _eResult                := E_PROGRESS.PROGRESS_ERROR;
      ELSE
        _eResult                := Enable(TRUE);
      END_IF

    E_INSTANCE_STATE.WORKING:
      IF NOT (_XtsTransportState.XpuState.DcLink) OR
         NOT (_XtsTransportState.XpuInfo.AllPositionsValid)
      THEN
        _eResult                := E_PROGRESS.PROGRESS_ERROR;
      ELSE
        _eResult                := Work(TRUE);
      END_IF

    E_INSTANCE_STATE.PROCEEDING:
      IF NOT (_XtsTransportState.XpuState.DcLink) OR
         NOT (_XtsTransportState.XpuInfo.AllPositionsValid)
      THEN
        _eResult                := E_PROGRESS.PROGRESS_ERROR;
      ELSE
        _eResult                := Proceed(TRUE);
      END_IF

    E_INSTANCE_STATE.FINISH:
      IF NOT (_XtsTransportState.XpuState.DcLink) OR
         NOT (_XtsTransportState.XpuInfo.AllPositionsValid)
      THEN
        _eResult                := E_PROGRESS.PROGRESS_ERROR;
      ELSE
        _eResult                := Finish(TRUE);
      END_IF

    E_INSTANCE_STATE.CLEARED:
      _eResult                  := Clear(TRUE);


  ELSE
    _eResult                    := E_PROGRESS.PROGRESS_INVALID;
  END_CASE

END_CASE
_State.XtsTransportState        REF= _XtsTransportState;
_State.InstanceStates           REF= _InstanceState;


IF (_nTimeVariant <> _nTimeVariantOld) OR
   (_nTimeVariant = 0)
THEN
  _nTimeVariantOld              := _nTimeVariant;
  CASE _nTimeVariant
  OF
    0:
      _tProcess[E_INSTANCE.INFEED]           := T#800MS;
      _tProcess[E_INSTANCE.OUTFEED_ROBOT_R1] := T#800MS;
      _tProcess[E_INSTANCE.OUTFEED_ROBOT_R2] := T#800MS;
    1:
      _tProcess[E_INSTANCE.INFEED]           := T#600MS;
      _tProcess[E_INSTANCE.OUTFEED_ROBOT_R1] := T#800MS;
      _tProcess[E_INSTANCE.OUTFEED_ROBOT_R2] := T#800MS;
    2:
      _tProcess[E_INSTANCE.INFEED]           := T#600MS;
      _tProcess[E_INSTANCE.OUTFEED_ROBOT_R1] := T#700MS;
      _tProcess[E_INSTANCE.OUTFEED_ROBOT_R2] := T#700MS;
    3:
      _tProcess[E_INSTANCE.INFEED]           := T#700MS;
      _tProcess[E_INSTANCE.OUTFEED_ROBOT_R1] := T#800MS;
      _tProcess[E_INSTANCE.OUTFEED_ROBOT_R2] := T#800MS;
    4:
      _tProcess[E_INSTANCE.INFEED]           := T#500MS;
      _tProcess[E_INSTANCE.OUTFEED_ROBOT_R1] := T#800MS;
      _tProcess[E_INSTANCE.OUTFEED_ROBOT_R2] := T#800MS;
    5:
      _tProcess[E_INSTANCE.INFEED]           := T#450MS;
      _tProcess[E_INSTANCE.OUTFEED_ROBOT_R1] := T#800MS;
      _tProcess[E_INSTANCE.OUTFEED_ROBOT_R2] := T#800MS;
  ELSE
      _tProcess[E_INSTANCE.INFEED]           := T#800MS;
      _tProcess[E_INSTANCE.OUTFEED_ROBOT_R1] := T#800MS;
      _tProcess[E_INSTANCE.OUTFEED_ROBOT_R2] := T#800MS;
  END_CASE
END_IF

_nAppState  := f_GetState(_State.AppState);
_nAppResult := f_GetProgress(_State.AppState);

_sAppState  := TO_STRING(_nAppState);
_sAppResult := TO_STRING(_nAppResult);

METHOD Check : BOOL // call this method in the extending/inheriting class
VAR
  _nIdx       : E_INSTANCE;
END_VAR
//-----------------------------------------------------------------------------
//-----------------------------------------------------------------------------
// reference checks
//-----------------------------------------------------------------------------
IF NOT __ISVALIDREF(_Ctrl)
THEN
  _eCheck                   := E_APP_CHECK.INVALID_CTRL_POINTER;
  RETURN;
END_IF

IF NOT __ISVALIDREF(_State)
THEN
  _eCheck                   := E_APP_CHECK.INVALID_STATE_POINTER;
  RETURN;
END_IF

IF NOT __ISVALIDREF(_XtsTransportCtrl)
THEN
  _eCheck                   := E_APP_CHECK.INVALID_TRANSPORT_CTRL_POINTER;
  RETURN;
END_IF

IF NOT __ISVALIDREF(_XtsTransportState)
THEN
  _eCheck                   := E_APP_CHECK.INVALID_TRANSPORT_STATE_POINTER;
  RETURN;
END_IF

IF NOT __ISVALIDREF(_InstanceCtrl)
THEN
  _eCheck                   := E_APP_CHECK.INVALID_INSTANCE_CONTROL_REFERENCE;
  RETURN;
END_IF

IF NOT __ISVALIDREF(_InstanceState)
THEN
  _eCheck                   := E_APP_CHECK.INVALID_INSTANCE_STATE_REFERENCE;
  RETURN;
END_IF
IF NOT __ISVALIDREF(_ItfProcessCollector)
THEN
  _eCheck                   := E_APP_CHECK.INVALID_COLLECTOR_INTERFACE;
  RETURN;
END_IF
IF NOT __ISVALIDREF(_ItfProcessList)
THEN
  _eCheck                   := E_APP_CHECK.INVALID_PROCESS_LIST_INTERFACE;
  RETURN;
END_IF
//-----------------------------------------------------------------------------
//-----------------------------------------------------------------------------
// interface checks
//-----------------------------------------------------------------------------
FOR _nIdx := 1 TO MAX_PROCESS
DO
  IF NOT (_ItfProcessCollector[_nIdx] <> 0) 
  THEN
    _eCheck                 := E_APP_CHECK.INVALID_COLLECTOR_INTERFACE;
    RETURN;
  END_IF
  
  IF NOT (_ItfProcessCollector[_nIdx].ProcessId > 0)
  THEN
    _eCheck                 := E_APP_CHECK.INVALID_PROCESS_LIST_INTERFACE;
    RETURN;
  END_IF
END_FOR
//-----------------------------------------------------------------------------
//-----------------------------------------------------------------------------
_eCheck                     := E_APP_CHECK.CHECK_DONE;
Check                       := TRUE;
END_METHOD

METHOD Clear : E_PROGRESS
VAR_INPUT
  Execute     : BOOL;
END_VAR
VAR_INST
  _nErrorId   : UDINT;
  _eState     : E_PROGRESS;

  _eInstance  : E_INSTANCE;
END_VAR
//-----------------------------------------------------------------------------
IF NOT Execute 
THEN 
	_eState                                         := E_PROGRESS.PROGRESS_INIT; 
END_IF 
//-----------------------------------------------------------------------------
IF NOT Check() 
THEN 
	Clear                                            := E_PROGRESS.PROGRESS_ERROR; 
	RETURN; 
END_IF
//-----------------------------------------------------------------------------
//-----------------------------------------------------------------------------
CASE _eState
OF
  //---------------------------------------------------------------------------------------------------------------
  //---------------------------------------------------------------------------------------------------------------
  E_PROGRESS.PROGRESS_INIT:                   // startup procedure for your application
    IF Execute
    THEN
      ListData(FALSE, TRUE);
      _eState                                             := E_PROGRESS.PROGRESS_BUSY;
  
      FOR _eInstance := E_INSTANCE.BUFFER_INFEED TO E_INSTANCE.SENDER_BUFFER_INFEED
      DO
        _InstanceCtrl[_eInstance].Cmd                     := E_INSTANCE_CMD.NULL;
      END_FOR
  
      IF (_MessageLevel > E_MessageType.eMessageError)
      THEN
        _stMsg.eType                                      := E_MessageType.eMessageInfo;
        _stMsg.eSubdevice                                 := e_Subdevice.Application_Clear;
        _stMsg.iErrorNumber                               := 0;
        _stMsg.sText                                      := concat(TO_STRING(_eState), ': ');
        f_MessageSet(_stMsg);
      END_IF
    END_IF

  //---------------------------------------------------------------------------------------------------------------
  //---------------------------------------------------------------------------------------------------------------
  E_PROGRESS.PROGRESS_BUSY:
    ListData(FALSE, FALSE);
    _InstanceCtrl[E_INSTANCE.BUFFER_INFEED].Cmd           := E_INSTANCE_CMD.INIT;
    //-----------------------------------------------------------------------------------
    CASE _InstanceState[E_INSTANCE.BUFFER_INFEED].State
    OF
      E_INSTANCE_STATE.DISABLED:
        CASE _InstanceState[E_INSTANCE.BUFFER_INFEED].Progress
        OF
          E_PROGRESS.PROGRESS_BUSY:           // check for startup to be done
            _InstanceCtrl[E_INSTANCE.BUFFER_INFEED].Cmd   := E_INSTANCE_CMD.DISABLE;
            _eState                                       := E_PROGRESS.PROGRESS_PREPARE; // go check next insatnce

            IF (_MessageLevel > E_MessageType.eMessageError)
            THEN
              _stMsg.eType          := E_MessageType.eMessageInfo;
              _stMsg.eSubdevice     := e_Subdevice.Application_Clear;
              _stMsg.iErrorNumber   := 0;
              _stMsg.sText          := concat(TO_STRING(E_INSTANCE.BUFFER_INFEED), ': cleared');
              f_MessageSet(_stMsg);
            END_IF
        END_CASE
    END_CASE

  //---------------------------------------------------------------------------------------------------------------
  //---------------------------------------------------------------------------------------------------------------
  E_PROGRESS.PROGRESS_PREPARE:
    _InstanceCtrl[E_INSTANCE.INFEED].Cmd                  := E_INSTANCE_CMD.INIT;
    //-----------------------------------------------------------------------------------
    CASE _InstanceState[E_INSTANCE.INFEED].State
    OF
      E_INSTANCE_STATE.DISABLED:
        CASE _InstanceState[E_INSTANCE.INFEED].Progress
        OF
          E_PROGRESS.PROGRESS_BUSY:           // check for startup to be done
          _InstanceCtrl[E_INSTANCE.INFEED].Cmd            := E_INSTANCE_CMD.DISABLE;
          _eState                                         := E_PROGRESS.PROGRESS_STARTUP; // go check next insatnce

          IF (_MessageLevel > E_MessageType.eMessageError)
          THEN
            _stMsg.eType          := E_MessageType.eMessageInfo;
            _stMsg.eSubdevice     := e_Subdevice.Application_Clear;
            _stMsg.iErrorNumber   := 0;
            _stMsg.sText          := concat(TO_STRING(E_INSTANCE.INFEED), ': cleared');
            f_MessageSet(_stMsg);
          END_IF
        END_CASE
    END_CASE

  //---------------------------------------------------------------------------------------------------------------
  //---------------------------------------------------------------------------------------------------------------
  E_PROGRESS.PROGRESS_STARTUP:
    _InstanceCtrl[E_INSTANCE.BUFFER_OUTFEED_ROBOT].Cmd    := E_INSTANCE_CMD.INIT;
    //-----------------------------------------------------------------------------------
    CASE _InstanceState[E_INSTANCE.BUFFER_OUTFEED_ROBOT].State
    OF
      E_INSTANCE_STATE.DISABLED:
        CASE _InstanceState[E_INSTANCE.BUFFER_OUTFEED_ROBOT].Progress
        OF
          E_PROGRESS.PROGRESS_BUSY:           // check for startup to be done
          _InstanceCtrl[E_INSTANCE.BUFFER_OUTFEED_ROBOT].Cmd   := E_INSTANCE_CMD.DISABLE;
          _eState                                         := E_PROGRESS.PROGRESS_CHECK; // go check next insatnce

          IF (_MessageLevel > E_MessageType.eMessageError)
          THEN
            _stMsg.eType          := E_MessageType.eMessageInfo;
            _stMsg.eSubdevice     := e_Subdevice.Application_Clear;
            _stMsg.iErrorNumber   := 0;
            _stMsg.sText          := concat(TO_STRING(E_INSTANCE.BUFFER_OUTFEED_ROBOT), ': cleared');
            f_MessageSet(_stMsg);
          END_IF
        END_CASE
    END_CASE

  //---------------------------------------------------------------------------------------------------------------
  //---------------------------------------------------------------------------------------------------------------
  E_PROGRESS.PROGRESS_CHECK:
    _InstanceCtrl[E_INSTANCE.OUTFEED_ROBOT_R1].Cmd        := E_INSTANCE_CMD.INIT;
    //-----------------------------------------------------------------------------------
    CASE _InstanceState[E_INSTANCE.OUTFEED_ROBOT_R1].State
    OF
      E_INSTANCE_STATE.DISABLED:
        CASE _InstanceState[E_INSTANCE.OUTFEED_ROBOT_R1].Progress
        OF
          E_PROGRESS.PROGRESS_BUSY:           // check for startup to be done
          _InstanceCtrl[E_INSTANCE.OUTFEED_ROBOT_R1].Cmd  := E_INSTANCE_CMD.DISABLE;
          _eState                                         := E_PROGRESS.PROGRESS_OCCUPIED; // go check next insatnce

          IF (_MessageLevel > E_MessageType.eMessageError)
          THEN
            _stMsg.eType          := E_MessageType.eMessageInfo;
            _stMsg.eSubdevice     := e_Subdevice.Application_Clear;
            _stMsg.iErrorNumber   := 0;
            _stMsg.sText          := concat(TO_STRING(E_INSTANCE.OUTFEED_ROBOT_R1), ': cleared');
            f_MessageSet(_stMsg);
          END_IF
        END_CASE
    END_CASE

  //---------------------------------------------------------------------------------------------------------------
  //---------------------------------------------------------------------------------------------------------------
  E_PROGRESS.PROGRESS_OCCUPIED:
    _InstanceCtrl[E_INSTANCE.OUTFEED_ROBOT_R2].Cmd        := E_INSTANCE_CMD.INIT;
    //-----------------------------------------------------------------------------------
    CASE _InstanceState[E_INSTANCE.OUTFEED_ROBOT_R2].State
    OF
      E_INSTANCE_STATE.DISABLED:
        CASE _InstanceState[E_INSTANCE.OUTFEED_ROBOT_R2].Progress
        OF
          E_PROGRESS.PROGRESS_BUSY:           // check for startup to be done
          _InstanceCtrl[E_INSTANCE.OUTFEED_ROBOT_R2].Cmd  := E_INSTANCE_CMD.DISABLE;
          _eState                                         := E_PROGRESS.PROGRESS_WORKING; // go check next insatnce

          IF (_MessageLevel > E_MessageType.eMessageError)
          THEN
            _stMsg.eType          := E_MessageType.eMessageInfo;
            _stMsg.eSubdevice     := e_Subdevice.Application_Clear;
            _stMsg.iErrorNumber   := 0;
            _stMsg.sText          := concat(TO_STRING(E_INSTANCE.OUTFEED_ROBOT_R2), ': cleared');
            f_MessageSet(_stMsg);
          END_IF
        END_CASE
    END_CASE

  //---------------------------------------------------------------------------------------------------------------
  //---------------------------------------------------------------------------------------------------------------
  E_PROGRESS.PROGRESS_WORKING:
    _InstanceCtrl[E_INSTANCE.SENDER_FAST].Cmd             := E_INSTANCE_CMD.INIT;
    //-----------------------------------------------------------------------------------
    CASE _InstanceState[E_INSTANCE.SENDER_FAST].State
    OF
      E_INSTANCE_STATE.DISABLED:
        CASE _InstanceState[E_INSTANCE.SENDER_FAST].Progress
        OF
          E_PROGRESS.PROGRESS_BUSY:           // check for startup to be done
          _InstanceCtrl[E_INSTANCE.SENDER_FAST].Cmd       := E_INSTANCE_CMD.DISABLE;
          _eState                                         := E_PROGRESS.PROGRESS_STILL_WORKING; // go check next insatnce

          IF (_MessageLevel > E_MessageType.eMessageError)
          THEN
            _stMsg.eType          := E_MessageType.eMessageInfo;
            _stMsg.eSubdevice     := e_Subdevice.Application_Clear;
            _stMsg.iErrorNumber   := 0;
            _stMsg.sText          := concat(TO_STRING(E_INSTANCE.SENDER_FAST), ': cleared');
            f_MessageSet(_stMsg);
          END_IF
        END_CASE
    END_CASE

  //---------------------------------------------------------------------------------------------------------------
  //---------------------------------------------------------------------------------------------------------------
  E_PROGRESS.PROGRESS_STILL_WORKING:
    _InstanceCtrl[E_INSTANCE.SENDER_BUFFER_INFEED].Cmd    := E_INSTANCE_CMD.INIT;
    //-----------------------------------------------------------------------------------
    CASE _InstanceState[E_INSTANCE.SENDER_BUFFER_INFEED].State
    OF
      E_INSTANCE_STATE.DISABLED:
        CASE _InstanceState[E_INSTANCE.SENDER_BUFFER_INFEED].Progress
        OF
          E_PROGRESS.PROGRESS_BUSY:           // check for startup to be done
          _InstanceCtrl[E_INSTANCE.SENDER_BUFFER_INFEED].Cmd    := E_INSTANCE_CMD.DISABLE;
          _eState                                         := E_PROGRESS.PROGRESS_DONE;

          IF (_MessageLevel > E_MessageType.eMessageError)
          THEN
            _stMsg.eType          := E_MessageType.eMessageInfo;
            _stMsg.eSubdevice     := e_Subdevice.Application_Clear;
            _stMsg.iErrorNumber   := 0;
            _stMsg.sText          := concat(TO_STRING(E_INSTANCE.SENDER_BUFFER_INFEED), ': cleared');
            f_MessageSet(_stMsg);
          END_IF

          IF (_MessageLevel > E_MessageType.eMessageError)
          THEN
            _stMsg.eType          := E_MessageType.eMessageInfo;
            _stMsg.eSubdevice     := e_Subdevice.Application_Clear;
            _stMsg.iErrorNumber   := 0;
            _stMsg.sText          := concat(TO_STRING(_eState), ': ');
            f_MessageSet(_stMsg);
          END_IF
        END_CASE
    END_CASE
END_CASE
//-----------------------------------------------------------------------------
//-----------------------------------------------------------------------------

Clear                                              := _eState;
END_METHOD

METHOD PRIVATE Cmd : E_INSTANCE_STATE
VAR_INPUT
  Command   : E_INSTANCE_CMD;
END_VAR
VAR_INST
  _eRslt    : E_PROGRESS;
  _eState   : E_INSTANCE_STATE;
END_VAR
IF NOT Check() THEN RETURN; END_IF


CASE Command
OF
  E_INSTANCE_CMD.NULL:  // clear all method calls
    _eState               := E_INSTANCE_STATE.NULL;
    _eRslt                := Init    (FALSE);
    _eRslt                := Disable (FALSE);
    _eRslt                := Enable  (FALSE);
    _eRslt                := Work    (FALSE);
    _eRslt                := Proceed (FALSE);
    _eRslt                := Finish  (FALSE);
    _eRslt                := Clear   (FALSE);

  E_INSTANCE_CMD.INIT:  // clear methods for initialization
    _eState               := E_INSTANCE_STATE.INIT;
    _eResult              := Init(FALSE);

ELSE
  IF NOT (_eInit = E_PROGRESS.PROGRESS_DONE)
  THEN
    // no init, no further commands possible
    _eState               := E_INSTANCE_STATE.INVALID;
  ELSE
    CASE Command
    OF
      E_INSTANCE_CMD.DISABLE:
        _eState           := E_INSTANCE_STATE.DISABLED;
        _eResult          := Disable (FALSE);

      E_INSTANCE_CMD.ENABLE:
        _eState           := E_INSTANCE_STATE.ENABLED;
        _eResult          := Enable  (FALSE);

      E_INSTANCE_CMD.WORK:
        _eState           := E_INSTANCE_STATE.WORKING;
        _eResult          := Work    (FALSE);

      E_INSTANCE_CMD.PROCEED:
        _eState           := E_INSTANCE_STATE.PROCEEDING;
        _eResult          := Proceed (FALSE);

      E_INSTANCE_CMD.FINISH:
        _eState           := E_INSTANCE_STATE.FINISH;
        _eResult          := Finish  (FALSE);

      E_INSTANCE_CMD.CLEAR:
        _eState           := E_INSTANCE_STATE.CLEARED;
        _eResult          := Clear   (FALSE);

    ELSE
        _eState           := E_INSTANCE_STATE.INVALID;
    END_CASE
  END_IF
END_CASE

Cmd                       := _eState;
END_METHOD

PROPERTY CollectorInterface : REFERENCE TO ARRAY[1..MAX_PROCESS] OF I_ProcessCollector
SET
_ItfProcessCollector REF= CollectorInterface;
END_SET
END_PROPERTY

PROPERTY Ctrl : REFERENCE TO ST_APP_CTRL
SET
_Ctrl REF= Ctrl;
END_SET
END_PROPERTY

METHOD Disable : E_PROGRESS // RemoveAllAxis from CA Group, disable CA Group, disable all movers
VAR_INPUT
  Execute     : BOOL;
END_VAR
VAR_INST
  _nErrorId   : UDINT;
  _eState     : E_PROGRESS;
END_VAR
//-----------------------------------------------------------------------------
IF NOT Execute 
THEN 
	_eState                       := E_PROGRESS.PROGRESS_INIT; 
END_IF 
//-----------------------------------------------------------------------------
IF NOT Check() 
THEN 
	Disable                       := E_PROGRESS.PROGRESS_ERROR; 
	RETURN; 
END_IF
//-----------------------------------------------------------------------------
//-----------------------------------------------------------------------------
CASE _eState
OF
  E_PROGRESS.PROGRESS_INIT:
    IF Execute
    THEN
      _nErrorId                 := 0;

      _XtsTransportCtrl.Cmd     := E_XTS_TRANSPORT_CTRL.CMD_NULL;
      _eState                   := E_PROGRESS.PROGRESS_BUSY;

      IF (_MessageLevel > E_MessageType.eMessageError)
      THEN
        _stMsg.eType            := E_MessageType.eMessageInfo;
        _stMsg.eSubdevice       := e_Subdevice.Application_Disable;
        _stMsg.iErrorNumber     := 0;
        _stMsg.sText            := concat(TO_STRING(_eState), ': ');
        f_MessageSet(_stMsg);
      END_IF
    END_IF

  E_PROGRESS.PROGRESS_BUSY:
    _XtsTransportCtrl.Cmd       := E_XTS_TRANSPORT_CTRL.CMD_GROUP_CLEAR; 
    _eState                     := E_PROGRESS.PROGRESS_PREPARE;
END_CASE
//-----------------------------------------------------------------------------
//-----------------------------------------------------------------------------
CASE _eState
OF
  E_PROGRESS.PROGRESS_PREPARE:
    IF (_XtsTransportState.State = E_XTS_TRANSPORT_STATE.TRANSPORT_GROUP_CLEAR + E_PROGRESS.PROGRESS_ERROR)
    THEN
      _eState                   := E_PROGRESS.PROGRESS_BUSY;
      _XtsTransportCtrl.Cmd     := E_XTS_TRANSPORT_CTRL.CMD_NULL;

      _nErrorId                 := _XtsTransportState.GroupInfo.GroupErrorId; 

    ELSIF (_XtsTransportState.State = E_XTS_TRANSPORT_STATE.TRANSPORT_GROUP_CLEAR + E_PROGRESS.PROGRESS_DONE)
    THEN
      _eState                   := E_PROGRESS.PROGRESS_STARTUP;

    END_IF
END_CASE
//-----------------------------------------------------------------------------
//-----------------------------------------------------------------------------
CASE _eState
OF
  E_PROGRESS.PROGRESS_STARTUP:
    _XtsTransportCtrl.Cmd       := E_XTS_TRANSPORT_CTRL.CMD_MOVER_DISABLE; 
    _eState                     := E_PROGRESS.PROGRESS_CHECK;
END_CASE
//-----------------------------------------------------------------------------
//-----------------------------------------------------------------------------
CASE _eState
OF
  E_PROGRESS.PROGRESS_CHECK:
    IF (_XtsTransportState.State = E_XTS_TRANSPORT_STATE.TRANSPORT_MOVER_DISABLE + E_PROGRESS.PROGRESS_ERROR)
    THEN
      _eState                   := E_PROGRESS.PROGRESS_BUSY;
      _XtsTransportCtrl.Cmd     := E_XTS_TRANSPORT_CTRL.CMD_NULL;

    ELSIF (_XtsTransportState.State = E_XTS_TRANSPORT_STATE.TRANSPORT_MOVER_DISABLE + E_PROGRESS.PROGRESS_DONE)
    THEN
      _eState                   := E_PROGRESS.PROGRESS_DONE;

      IF (_MessageLevel > E_MessageType.eMessageError)
      THEN
        _stMsg.eType            := E_MessageType.eMessageInfo;
        _stMsg.eSubdevice       := e_Subdevice.Application_Disable;
        _stMsg.iErrorNumber     := 0;
        _stMsg.sText            := concat(TO_STRING(_eState), ': ');
        f_MessageSet(_stMsg);
      END_IF
    END_IF
END_CASE
//-----------------------------------------------------------------------------
//-----------------------------------------------------------------------------

Disable                         := _eState;
END_METHOD

METHOD Enable : E_PROGRESS // AddAllAxis to CA Group, Enable CA Group, Enable all movers
VAR_INPUT
  Execute     : BOOL;
END_VAR
VAR_INST
  _nErrorId   : UDINT;
  _eState     : E_PROGRESS;
END_VAR
//-----------------------------------------------------------------------------
IF NOT Execute 
THEN 
	_eState                       := E_PROGRESS.PROGRESS_INIT; 
END_IF 
//-----------------------------------------------------------------------------
IF NOT Check() 
THEN 
	Enable                        := E_PROGRESS.PROGRESS_ERROR; 
	RETURN; 
END_IF
//-----------------------------------------------------------------------------
//-----------------------------------------------------------------------------
CASE _eState
OF
  E_PROGRESS.PROGRESS_INIT:
    IF Execute
    THEN
      _nErrorId                 := 0;

      _XtsTransportCtrl.Cmd     := E_XTS_TRANSPORT_CTRL.CMD_NULL;
      _eState                   := E_PROGRESS.PROGRESS_BUSY;

      IF (_MessageLevel > E_MessageType.eMessageError)
      THEN
        _stMsg.eType            := E_MessageType.eMessageInfo;
        _stMsg.eSubdevice       := e_Subdevice.Application_Enable;
        _stMsg.iErrorNumber     := 0;
        _stMsg.sText            := concat(TO_STRING(_eState), ': ');
        f_MessageSet(_stMsg);
      END_IF
    END_IF

  E_PROGRESS.PROGRESS_BUSY:
    _XtsTransportCtrl.Cmd       := E_XTS_TRANSPORT_CTRL.CMD_GROUP_BUILD; 
    _eState                     := E_PROGRESS.PROGRESS_PREPARE;
END_CASE
//-----------------------------------------------------------------------------
//-----------------------------------------------------------------------------
CASE _eState
OF
  E_PROGRESS.PROGRESS_PREPARE:
    IF (_XtsTransportState.State = E_XTS_TRANSPORT_STATE.TRANSPORT_GROUP_BUILD + E_PROGRESS.PROGRESS_ERROR)
    THEN
      _eState                   := E_PROGRESS.PROGRESS_STILL_WORKING;
      _nErrorId                 := _XtsTransportState.GroupInfo.GroupErrorId;
      _XtsTransportCtrl.Cmd     := E_XTS_TRANSPORT_CTRL.CMD_GROUP_CLEAR; 

    ELSIF (_XtsTransportState.State = E_XTS_TRANSPORT_STATE.TRANSPORT_GROUP_BUILD + E_PROGRESS.PROGRESS_DONE)
    THEN
      _eState                   := E_PROGRESS.PROGRESS_STARTUP;
    END_IF
END_CASE
//-----------------------------------------------------------------------------
//-----------------------------------------------------------------------------
CASE _eState
OF
  E_PROGRESS.PROGRESS_STARTUP:
    IF (_XtsTransportState.XpuState.DcLink)
    THEN
      _XtsTransportCtrl.Cmd     := E_XTS_TRANSPORT_CTRL.CMD_MOVER_ENABLE; 
      _eState                   := E_PROGRESS.PROGRESS_CHECK;
    END_IF
END_CASE
//-----------------------------------------------------------------------------
//-----------------------------------------------------------------------------
CASE _eState
OF
  E_PROGRESS.PROGRESS_CHECK:
    IF (_XtsTransportState.State = E_XTS_TRANSPORT_STATE.TRANSPORT_MOVER_ENABLE + E_PROGRESS.PROGRESS_ERROR)
    THEN
      _eState                   := E_PROGRESS.PROGRESS_ERROR;

    ELSIF (_XtsTransportState.State = E_XTS_TRANSPORT_STATE.TRANSPORT_MOVER_ENABLE + E_PROGRESS.PROGRESS_DONE)
    THEN
      _eState                   := E_PROGRESS.PROGRESS_OCCUPIED;
    END_IF
END_CASE
//-----------------------------------------------------------------------------
//-----------------------------------------------------------------------------
CASE _eState
OF
  E_PROGRESS.PROGRESS_OCCUPIED:
    _XtsTransportCtrl.Cmd       := E_XTS_TRANSPORT_CTRL.CMD_GROUP_ENABLE; 
    _eState                     := E_PROGRESS.PROGRESS_WORKING;
END_CASE
//-----------------------------------------------------------------------------
//-----------------------------------------------------------------------------
CASE _eState
OF
  E_PROGRESS.PROGRESS_WORKING:
    IF (_XtsTransportState.State = E_XTS_TRANSPORT_STATE.TRANSPORT_GROUP_ENABLE + E_PROGRESS.PROGRESS_ERROR)
    THEN
      _eState                   := E_PROGRESS.PROGRESS_ERROR;

    ELSIF (_XtsTransportState.State = E_XTS_TRANSPORT_STATE.TRANSPORT_GROUP_ENABLE + E_PROGRESS.PROGRESS_DONE)
    THEN
      _eState                   := E_PROGRESS.PROGRESS_DONE;

      IF (_MessageLevel > E_MessageType.eMessageError)
      THEN
        _stMsg.eType            := E_MessageType.eMessageInfo;
        _stMsg.eSubdevice       := e_Subdevice.Application_Enable;
        _stMsg.iErrorNumber     := 0;
        _stMsg.sText            := concat(TO_STRING(_eState), ': ');
        f_MessageSet(_stMsg);
      END_IF
    END_IF
END_CASE
//-----------------------------------------------------------------------------
//-----------------------------------------------------------------------------
CASE _eState
OF
  E_PROGRESS.PROGRESS_STILL_WORKING:
    IF (_XtsTransportState.State = E_XTS_TRANSPORT_STATE.TRANSPORT_GROUP_CLEAR + E_PROGRESS.PROGRESS_ERROR)
    THEN
      _eState                   := E_PROGRESS.PROGRESS_ERROR;
      _nErrorId                 := _XtsTransportState.GroupInfo.GroupErrorId;

    ELSIF (_XtsTransportState.State = E_XTS_TRANSPORT_STATE.TRANSPORT_GROUP_CLEAR + E_PROGRESS.PROGRESS_DONE)
    THEN
      _eState                   := E_PROGRESS.PROGRESS_BUSY;
    END_IF
END_CASE
//-----------------------------------------------------------------------------
//-----------------------------------------------------------------------------

Enable                          := _eState;
END_METHOD

METHOD Finish : E_PROGRESS
VAR_INPUT
  Execute     : BOOL;
END_VAR
VAR_INST
  _nErrorId               : UDINT;
  _eState                 : E_PROGRESS;

  _nExp                   : BYTE;
  _WriteData              : ST_PROCESS_DATA;
  _ListResult             : ST_PROCESS_LIST_RESULT;

  _eInst                  : E_INSTANCE;
  _bDbg : BOOL;
  {attribute 'displaymode':='bin'}
  _wDisable               : T_PROCESS;

  _nSwitch                : UINT;
  _TransportState         : E_XTS_TRANSPORT_STATE;
  _JobResult              : E_PROGRESS;
END_VAR
//-----------------------------------------------------------------------------
IF NOT Execute 
THEN 
	_eState                       := E_PROGRESS.PROGRESS_INIT; 
END_IF 
//-----------------------------------------------------------------------------
IF NOT Check() 
THEN 
	Finish                        := E_PROGRESS.PROGRESS_ERROR; 
	RETURN; 
END_IF
//-----------------------------------------------------------------------------
//-----------------------------------------------------------------------------
CASE _eState
OF
  E_PROGRESS.PROGRESS_INIT:
    IF Execute
    THEN
      _nErrorId                 := 0;
      _JobResult                := ListData(TRUE, FALSE);     // reset simulated transfersystem

      IF NOT (_XtsTransportState.GroupInfo.GroupErrorStop)
      THEN
        _eState                 := E_PROGRESS.PROGRESS_BUSY;

        IF (_MessageLevel > E_MessageType.eMessageError)
        THEN
          _stMsg.eType          := E_MessageType.eMessageInfo;
          _stMsg.eSubdevice     := e_Subdevice.Application_Finish;
          _stMsg.iErrorNumber   := 0;
          _stMsg.sText          := concat(TO_STRING(_eState), ': ');
          f_MessageSet(_stMsg);
        END_IF
      ELSE
        _nErrorId               := _XtsTransportState.GroupInfo.GroupErrorId;
        _eState                 := E_PROGRESS.PROGRESS_ERROR;

        _stMsg.eType            := E_MessageType.eMessageError;
        _stMsg.eSubdevice       := e_Subdevice.Application_Finish;
        _stMsg.iErrorNumber     := _nErrorId;
        _stMsg.sText            := concat(TO_STRING(_eState), ': ');
        _stMsg.sText            := concat(_stMsg.sText, ' CaGroup ErrorStop');
        f_MessageSet(_stMsg);
      END_IF
    END_IF


  E_PROGRESS.PROGRESS_BUSY:
    IF (_XtsTransportState.State = E_XTS_TRANSPORT_STATE.TRANSPORT_START   + E_PROGRESS.PROGRESS_ERROR) OR
       (_XtsTransportState.State = E_XTS_TRANSPORT_STATE.TRANSPORT_RESTART + E_PROGRESS.PROGRESS_ERROR)
    THEN
      _eState                   := E_PROGRESS.PROGRESS_ERROR;

      _stMsg.eType              := E_MessageType.eMessageError;
      _stMsg.eSubdevice         := e_Subdevice.Application_Finish;
      _stMsg.iErrorNumber       := 0;
      _stMsg.sText              := concat(TO_STRING(_eState), ': ');
      _stMsg.sText              := concat(_stMsg.sText, TO_STRING(_XtsTransportState.State MOD E_PROGRESS.PROGRESS_ERROR));
      f_MessageSet(_stMsg);

    ELSIF (_XtsTransportState.State = E_XTS_TRANSPORT_STATE.TRANSPORT_START   + E_PROGRESS.PROGRESS_DONE) OR
          (_XtsTransportState.State = E_XTS_TRANSPORT_STATE.TRANSPORT_RESTART + E_PROGRESS.PROGRESS_DONE)
    THEN
      _JobResult                := ListData(FALSE, FALSE);     // stop simulated transfersystem
      _wDisable                 := 0;
      _eState                   := E_PROGRESS.PROGRESS_PREPARE;

      IF (_MessageLevel > E_MessageType.eMessageError)
      THEN
        _stMsg.eType            := E_MessageType.eMessageInfo;
        _stMsg.eSubdevice       := e_Subdevice.Application_Finish;
        _stMsg.iErrorNumber     := 0;
        _stMsg.sText            := concat(TO_STRING(_eState), ': ');
        _stMsg.sText            := concat(_stMsg.sText, TO_STRING(_XtsTransportState.State MOD E_PROGRESS.PROGRESS_DONE));
        f_MessageSet(_stMsg);
      END_IF
    END_IF
END_CASE
//-----------------------------------------------------------------------------
//-----------------------------------------------------------------------------
CASE _eState
OF
  E_PROGRESS.PROGRESS_PREPARE:  // SENDER_BUFFER_INFEED sends movers to BUFFER_INFEED
                                //  - this instance has to stop first
    CASE _InstanceState[E_INSTANCE.SENDER_BUFFER_INFEED].State
    OF
    E_INSTANCE_STATE.DISABLED:

      CASE _InstanceState[E_INSTANCE.SENDER_BUFFER_INFEED].Progress
      OF
      E_PROGRESS.PROGRESS_BUSY,
      E_PROGRESS.PROGRESS_PREPARE:
        _eState                                               := E_PROGRESS.PROGRESS_STARTUP;
        _InstanceCtrl[E_INSTANCE.SENDER_BUFFER_INFEED].Cmd    := E_INSTANCE_CMD.DISABLE;
  
        _wDisable                                             := _ItfProcessCollector[E_INSTANCE.SENDER_BUFFER_INFEED].
                                                                 SetBit(_wDisable, TO_BYTE(E_INSTANCE.SENDER_BUFFER_INFEED-1));
        IF (_MessageLevel > E_MessageType.eMessageError)
        THEN
          _stMsg.eType                                        := E_MessageType.eMessageInfo;
          _stMsg.eSubdevice                                   := e_Subdevice.Application_Finish;
          _stMsg.iErrorNumber                                 := 0;
          _stMsg.sText                                        := concat(TO_STRING(E_INSTANCE.SENDER_BUFFER_INFEED), ': _wDisable  ');
          _stMsg.sText                                        := concat(_stMsg.sText, _ItfProcessCollector[E_INSTANCE.SENDER_BUFFER_INFEED].BitsToString(_wDisable));
          f_MessageSet(_stMsg);
        END_IF
      END_CASE
    END_CASE
END_CASE
//-----------------------------------------------------------------------------
//-----------------------------------------------------------------------------
CASE _eState
OF
  E_PROGRESS.PROGRESS_STARTUP:
    _JobResult                                                := ListData(FALSE, FALSE);     // stop simulated transfersystem

    CASE _InstanceState[E_INSTANCE.BUFFER_INFEED].State
    OF
    E_INSTANCE_STATE.DISABLED,
    E_INSTANCE_STATE.DETECT_IN_LIST:

      _eState                                                 := E_PROGRESS.PROGRESS_CHECK;
      _InstanceCtrl[E_INSTANCE.BUFFER_INFEED].Cmd             := E_INSTANCE_CMD.DISABLE;
  
      IF NOT (_ItfProcessCollector[E_INSTANCE.BUFFER_INFEED].GetBit(_wDisable, TO_BYTE(E_INSTANCE.BUFFER_INFEED-1)))
      THEN
        _wDisable                                             := _ItfProcessCollector[E_INSTANCE.BUFFER_INFEED].
                                                                 SetBit(_wDisable, TO_BYTE(E_INSTANCE.BUFFER_INFEED-1));
  
        IF (_MessageLevel > E_MessageType.eMessageError)
        THEN
          _stMsg.eType                                        := E_MessageType.eMessageInfo;
          _stMsg.eSubdevice                                   := e_Subdevice.Application_Finish;
          _stMsg.iErrorNumber                                 := 0;
          _stMsg.sText                                        := concat(TO_STRING(E_INSTANCE.BUFFER_INFEED), ': _wDisable  ');
          _stMsg.sText                                        := concat(_stMsg.sText, _ItfProcessCollector[E_INSTANCE.BUFFER_INFEED].BitsToString(_wDisable));
          f_MessageSet(_stMsg);
        END_IF
      END_IF

    E_INSTANCE_STATE.ENABLED:
      _InstanceCtrl[E_INSTANCE.BUFFER_INFEED].Cmd             := E_INSTANCE_CMD.DISABLE;


    E_INSTANCE_STATE.FINISH:
      CASE _InstanceState[E_INSTANCE.BUFFER_INFEED].Progress
      OF
        E_PROGRESS.PROGRESS_BUSY:
          _InstanceCtrl[E_INSTANCE.BUFFER_INFEED].Cmd         := E_INSTANCE_CMD.FINISH;

        E_PROGRESS.PROGRESS_OCCUPIED:
          _InstanceCtrl[E_INSTANCE.BUFFER_INFEED].Cmd         := E_INSTANCE_CMD.PROCEED;
      END_CASE
    END_CASE
END_CASE
//-----------------------------------------------------------------------------
//-----------------------------------------------------------------------------
CASE _eState
OF
  E_PROGRESS.PROGRESS_CHECK:
    CASE _InstanceState[E_INSTANCE.INFEED].State
    OF
    E_INSTANCE_STATE.DISABLED,
    E_INSTANCE_STATE.DETECT_IN_LIST:

      CASE _InstanceState[E_INSTANCE.INFEED].Progress
      OF
      E_PROGRESS.PROGRESS_BUSY:
          IF (_ItfProcessCollector[E_INSTANCE.BUFFER_INFEED].QueueProcessCount > 0)
          THEN
            _eState                                           := E_PROGRESS.PROGRESS_STARTUP;
            _InstanceCtrl[E_INSTANCE.INFEED].Cmd              := E_INSTANCE_CMD.ENABLE;

          ELSIF (_ItfProcessList[E_INSTANCE.INFEED].Count > 0)
          THEN
            _InstanceCtrl[E_INSTANCE.INFEED].Cmd              := E_INSTANCE_CMD.ENABLE;
          ELSE
            _eState                                           := E_PROGRESS.PROGRESS_OCCUPIED;
            _InstanceCtrl[E_INSTANCE.INFEED].Cmd              := E_INSTANCE_CMD.DISABLE;

            IF NOT (_ItfProcessCollector[E_INSTANCE.INFEED].GetBit(_wDisable, TO_BYTE(E_INSTANCE.INFEED-1)))
            THEN
              _wDisable                                       := _ItfProcessCollector[E_INSTANCE.INFEED].
                                                                   SetBit(_wDisable, TO_BYTE(E_INSTANCE.INFEED-1));

              IF (_MessageLevel > E_MessageType.eMessageError)
              THEN
                _stMsg.eType                                  := E_MessageType.eMessageInfo;
                _stMsg.eSubdevice                             := e_Subdevice.Application_Finish;
                _stMsg.iErrorNumber                           := 0;
                _stMsg.sText                                  := concat(TO_STRING(E_INSTANCE.INFEED), ': _wDisable ');
                _stMsg.sText                                  := concat(_stMsg.sText, _ItfProcessCollector[E_INSTANCE.INFEED].BitsToString(_wDisable));
                f_MessageSet(_stMsg);
              END_IF
            END_IF
          END_IF
      END_CASE

    E_INSTANCE_STATE.ENABLED:
      CASE _InstanceState[E_INSTANCE.INFEED].Progress
      OF
        E_PROGRESS.PROGRESS_OCCUPIED:
          _InstanceCtrl[E_INSTANCE.INFEED].Cmd                := E_INSTANCE_CMD.PROCEED;
      END_CASE


    E_INSTANCE_STATE.WORKING:
      CASE _InstanceState[E_INSTANCE.INFEED].Progress
      OF
        E_PROGRESS.PROGRESS_BUSY:
          _InstanceCtrl[E_INSTANCE.INFEED].Cmd                := E_INSTANCE_CMD.WORK;
          _tonProcess [E_INSTANCE.INFEED]
                                          (IN                 := FALSE, 
                                           PT                 := _tProcess[E_INSTANCE.INFEED]);
  
        E_PROGRESS.PROGRESS_CHECK:
          _tonProcess [E_INSTANCE.INFEED]
                                          (IN                 := TRUE, 
                                           PT                 := _tProcess[E_INSTANCE.INFEED]);
  
          IF _tonProcess [E_INSTANCE.INFEED].Q
          THEN
            _InstanceCtrl[E_INSTANCE.INFEED].Cmd              := E_INSTANCE_CMD.FINISH;
          END_IF
      END_CASE

    E_INSTANCE_STATE.FINISH:
      CASE _InstanceState[E_INSTANCE.INFEED].Progress
      OF
        E_PROGRESS.PROGRESS_BUSY:
          _InstanceCtrl[E_INSTANCE.INFEED].Cmd                := E_INSTANCE_CMD.FINISH;

        E_PROGRESS.PROGRESS_OCCUPIED:
          _InstanceCtrl[E_INSTANCE.INFEED].Cmd                := E_INSTANCE_CMD.PROCEED;
      END_CASE
    END_CASE

    CASE _InstanceState[E_INSTANCE.BUFFER_OUTFEED_ROBOT].State
    OF
    E_INSTANCE_STATE.DISABLED:

      CASE _InstanceState[E_INSTANCE.BUFFER_OUTFEED_ROBOT].Progress
      OF
      E_PROGRESS.PROGRESS_BUSY:
        _InstanceCtrl[E_INSTANCE.BUFFER_OUTFEED_ROBOT].Cmd    := E_INSTANCE_CMD.ENABLE;
      END_CASE

    E_INSTANCE_STATE.FINISH:
      CASE _InstanceState[E_INSTANCE.BUFFER_OUTFEED_ROBOT].Progress
      OF
        E_PROGRESS.PROGRESS_BUSY:
          _InstanceCtrl[E_INSTANCE.BUFFER_OUTFEED_ROBOT].Cmd  := E_INSTANCE_CMD.FINISH;

        E_PROGRESS.PROGRESS_OCCUPIED:
          _InstanceCtrl[E_INSTANCE.BUFFER_OUTFEED_ROBOT].Cmd  := E_INSTANCE_CMD.PROCEED;

        E_PROGRESS.PROGRESS_DONE:
          _InstanceCtrl[E_INSTANCE.BUFFER_OUTFEED_ROBOT].Cmd  := E_INSTANCE_CMD.DISABLE;
      END_CASE
    END_CASE

    CASE _InstanceState[E_INSTANCE.SENDER_FAST].State
    OF
      E_INSTANCE_STATE.DISABLED:
        CASE _InstanceState[E_INSTANCE.SENDER_FAST].Progress
        OF
          E_PROGRESS.PROGRESS_BUSY:
            IF NOT (_ItfProcessCollector[E_INSTANCE.OUTFEED_ROBOT_R1].QueueProcessCount < 12) OR 
               NOT (_ItfProcessCollector[E_INSTANCE.OUTFEED_ROBOT_R2].QueueProcessCount < 12)
            THEN
              _InstanceCtrl[E_INSTANCE.SENDER_FAST].Cmd       := E_INSTANCE_CMD.ENABLE;

            ELSIF (_ItfProcessCollector[E_INSTANCE.SENDER_FAST].QueueProcessCount > 0)
            THEN
              _InstanceCtrl[E_INSTANCE.SENDER_FAST].Cmd       := E_INSTANCE_CMD.ENABLE;
            ELSE
              _InstanceCtrl[E_INSTANCE.SENDER_FAST].Cmd       := E_INSTANCE_CMD.DISABLE;

              IF NOT (_ItfProcessCollector[E_INSTANCE.SENDER_FAST].GetBit(_wDisable, TO_BYTE(E_INSTANCE.SENDER_FAST-1)))
              THEN
                _wDisable                                     := _ItfProcessCollector[E_INSTANCE.SENDER_FAST].
                                                                 SetBit(_wDisable, TO_BYTE(E_INSTANCE.SENDER_FAST-1));
    
                IF (_MessageLevel > E_MessageType.eMessageError)
                THEN
                  _stMsg.eType                                := E_MessageType.eMessageInfo;
                  _stMsg.eSubdevice                           := e_Subdevice.Application_Finish;
                  _stMsg.iErrorNumber                         := 0;
                  _stMsg.sText                                := concat(TO_STRING(E_INSTANCE.SENDER_FAST), ': _wDisable ');
                  _stMsg.sText                                := concat(_stMsg.sText, _ItfProcessCollector[E_INSTANCE.SENDER_FAST].BitsToString(_wDisable));
                  f_MessageSet(_stMsg);
                END_IF
              END_IF
            END_IF
        END_CASE

      E_INSTANCE_STATE.FINISH:
        CASE _InstanceState[E_INSTANCE.SENDER_FAST].Progress
        OF
          E_PROGRESS.PROGRESS_BUSY:
            _InstanceCtrl[E_INSTANCE.SENDER_FAST].Cmd         := E_INSTANCE_CMD.FINISH;
        END_CASE
      END_CASE
END_CASE
//-----------------------------------------------------------------------------
//-----------------------------------------------------------------------------
CASE _eState
OF
  E_PROGRESS.PROGRESS_OCCUPIED:
    CASE _InstanceState[E_INSTANCE.BUFFER_OUTFEED_ROBOT].State
    OF
    E_INSTANCE_STATE.DISABLED:

      CASE _InstanceState[E_INSTANCE.BUFFER_OUTFEED_ROBOT].Progress
      OF
      E_PROGRESS.PROGRESS_BUSY:
        IF (_ItfProcessCollector[E_INSTANCE.INFEED].QueueProcessCount > 11)
        THEN
          _eState                                             := E_PROGRESS.PROGRESS_CHECK;
          _InstanceCtrl[E_INSTANCE.BUFFER_OUTFEED_ROBOT].Cmd  := E_INSTANCE_CMD.ENABLE;

        ELSIF (_ItfProcessCollector[E_INSTANCE.BUFFER_OUTFEED_ROBOT].QueueProcessCount > 0)
        THEN
          _InstanceCtrl[E_INSTANCE.BUFFER_OUTFEED_ROBOT].Cmd  := E_INSTANCE_CMD.ENABLE;
        ELSE
          _eState                                             := E_PROGRESS.PROGRESS_WORKING;
          _InstanceCtrl[E_INSTANCE.BUFFER_OUTFEED_ROBOT].Cmd  := E_INSTANCE_CMD.DISABLE;

            IF NOT (_ItfProcessCollector[E_INSTANCE.BUFFER_OUTFEED_ROBOT].GetBit(_wDisable, TO_BYTE(E_INSTANCE.BUFFER_OUTFEED_ROBOT-1)))
            THEN
              _wDisable                                       := _ItfProcessCollector[E_INSTANCE.BUFFER_OUTFEED_ROBOT].
                                                                   SetBit(_wDisable, TO_BYTE(E_INSTANCE.BUFFER_OUTFEED_ROBOT-1));

              IF (_MessageLevel > E_MessageType.eMessageError)
              THEN
                _stMsg.eType                                  := E_MessageType.eMessageInfo;
                _stMsg.eSubdevice                             := e_Subdevice.Application_Finish;
                _stMsg.iErrorNumber                           := 0;
                _stMsg.sText                                  := concat(TO_STRING(E_INSTANCE.BUFFER_OUTFEED_ROBOT), ': _wDisable ');
                _stMsg.sText                                  := concat(_stMsg.sText, _ItfProcessCollector[E_INSTANCE.BUFFER_OUTFEED_ROBOT].BitsToString(_wDisable));
                f_MessageSet(_stMsg);
              END_IF
            END_IF
        END_IF
      END_CASE

    E_INSTANCE_STATE.ENABLED:
      _InstanceCtrl[E_INSTANCE.BUFFER_OUTFEED_ROBOT].Cmd      := E_INSTANCE_CMD.DISABLE;


    E_INSTANCE_STATE.FINISH:
      CASE _InstanceState[E_INSTANCE.BUFFER_OUTFEED_ROBOT].Progress
      OF
        E_PROGRESS.PROGRESS_BUSY:
          _InstanceCtrl[E_INSTANCE.BUFFER_OUTFEED_ROBOT].Cmd  := E_INSTANCE_CMD.FINISH;

        E_PROGRESS.PROGRESS_OCCUPIED:
          _InstanceCtrl[E_INSTANCE.BUFFER_OUTFEED_ROBOT].Cmd  := E_INSTANCE_CMD.PROCEED;

        E_PROGRESS.PROGRESS_DONE:
          _InstanceCtrl[E_INSTANCE.BUFFER_OUTFEED_ROBOT].Cmd  := E_INSTANCE_CMD.DISABLE;
      END_CASE
    END_CASE
END_CASE
//-----------------------------------------------------------------------------
//-----------------------------------------------------------------------------
CASE _eState
OF
  E_PROGRESS.PROGRESS_WORKING:
    IF (_wDisable = EXPT(2, E_INSTANCE.SENDER_BUFFER_INFEED)-1)
    THEN
      _eState                                                 := E_PROGRESS.PROGRESS_STILL_WORKING;
    END_IF

    //-------------------------------------------------------------------------
    // E_INSTANCE.OUTFEED_ROBOT_R1
    //-------------------------------------------------------------------------
    CASE _InstanceState[E_INSTANCE.OUTFEED_ROBOT_R1].State
    OF
    E_INSTANCE_STATE.DISABLED:
      CASE _InstanceState[E_INSTANCE.OUTFEED_ROBOT_R1].Progress
      OF
      E_PROGRESS.PROGRESS_BUSY:
        IF (_ItfProcessCollector[E_INSTANCE.OUTFEED_ROBOT_R1].QueueProcessCount < 12)
        THEN
          _InstanceCtrl[E_INSTANCE.OUTFEED_ROBOT_R1].Cmd      := E_INSTANCE_CMD.DISABLE;
  
          IF NOT (_ItfProcessCollector[E_INSTANCE.OUTFEED_ROBOT_R1].GetBit(_wDisable, TO_BYTE(E_INSTANCE.OUTFEED_ROBOT_R1-1)))
          THEN
            _wDisable                                         := _ItfProcessCollector[E_INSTANCE.OUTFEED_ROBOT_R1].
                                                                 SetBit(_wDisable, TO_BYTE(E_INSTANCE.OUTFEED_ROBOT_R1-1));

            IF (_MessageLevel > E_MessageType.eMessageError)
            THEN
              _stMsg.eType                                    := E_MessageType.eMessageInfo;
              _stMsg.eSubdevice                               := e_Subdevice.Application_Finish;
              _stMsg.iErrorNumber                             := 0;
              _stMsg.sText                                    := concat(TO_STRING(E_INSTANCE.OUTFEED_ROBOT_R1), ': _wDisable ');
              _stMsg.sText                                    := concat(_stMsg.sText, _ItfProcessCollector[E_INSTANCE.OUTFEED_ROBOT_R1].BitsToString(_wDisable));
              f_MessageSet(_stMsg);
            END_IF
          END_IF
        ELSE
          _InstanceCtrl[E_INSTANCE.OUTFEED_ROBOT_R1].Cmd      := E_INSTANCE_CMD.ENABLE;
        END_IF
      END_CASE

      E_INSTANCE_STATE.ENABLED:
        CASE _InstanceState[E_INSTANCE.OUTFEED_ROBOT_R1].Progress
        OF
          E_PROGRESS.PROGRESS_OCCUPIED:
            _InstanceCtrl[E_INSTANCE.OUTFEED_ROBOT_R1].Cmd    := E_INSTANCE_CMD.PROCEED;
        END_CASE


      E_INSTANCE_STATE.WORKING:
        CASE _InstanceState[E_INSTANCE.OUTFEED_ROBOT_R1].Progress
        OF
          E_PROGRESS.PROGRESS_BUSY:
            _tonProcess [E_INSTANCE.OUTFEED_ROBOT_R1]
                                                  (IN         := FALSE, 
                                                   PT         := _tProcess[E_INSTANCE.OUTFEED_ROBOT_R1]);

            _InstanceCtrl[E_INSTANCE.OUTFEED_ROBOT_R1].Cmd    := E_INSTANCE_CMD.WORK;
    

          E_PROGRESS.PROGRESS_CHECK:
            _tonProcess [E_INSTANCE.OUTFEED_ROBOT_R1]
                                                  (IN         := TRUE, 
                                                   PT         := _tProcess[E_INSTANCE.OUTFEED_ROBOT_R1]);
    
            IF _tonProcess [E_INSTANCE.OUTFEED_ROBOT_R1].Q
            THEN
              _InstanceCtrl[E_INSTANCE.OUTFEED_ROBOT_R1].Cmd  := E_INSTANCE_CMD.FINISH;
            END_IF
        END_CASE

      E_INSTANCE_STATE.FINISH:
        CASE _InstanceState[E_INSTANCE.OUTFEED_ROBOT_R1].Progress
        OF
          E_PROGRESS.PROGRESS_BUSY:
            _InstanceCtrl[E_INSTANCE.OUTFEED_ROBOT_R1].Cmd    := E_INSTANCE_CMD.FINISH;

          E_PROGRESS.PROGRESS_DONE:
            _InstanceCtrl[E_INSTANCE.OUTFEED_ROBOT_R1].Cmd    := E_INSTANCE_CMD.DISABLE;
        END_CASE
      END_CASE

    //-------------------------------------------------------------------------
    // E_INSTANCE.OUTFEED_ROBOT_R2
    //-------------------------------------------------------------------------
    CASE _InstanceState[E_INSTANCE.OUTFEED_ROBOT_R2].State
    OF
    E_INSTANCE_STATE.DISABLED:
      CASE _InstanceState[E_INSTANCE.OUTFEED_ROBOT_R2].Progress
      OF
      E_PROGRESS.PROGRESS_BUSY:
        IF (_ItfProcessCollector[E_INSTANCE.OUTFEED_ROBOT_R2].QueueProcessCount < 12)
        THEN
          _InstanceCtrl[E_INSTANCE.OUTFEED_ROBOT_R2].Cmd      := E_INSTANCE_CMD.DISABLE;

          IF NOT (_ItfProcessCollector[E_INSTANCE.OUTFEED_ROBOT_R2].GetBit(_wDisable, TO_BYTE(E_INSTANCE.OUTFEED_ROBOT_R2-1)))
          THEN
            _wDisable                                         := _ItfProcessCollector[E_INSTANCE.OUTFEED_ROBOT_R2].
                                                                 SetBit(_wDisable, TO_BYTE(E_INSTANCE.OUTFEED_ROBOT_R2-1));

            IF (_MessageLevel > E_MessageType.eMessageError)
            THEN
              _stMsg.eType                                    := E_MessageType.eMessageInfo;
              _stMsg.eSubdevice                               := e_Subdevice.Application_Finish;
              _stMsg.iErrorNumber                             := 0;
              _stMsg.sText                                    := concat(TO_STRING(E_INSTANCE.OUTFEED_ROBOT_R2), ': _wDisable ');
              _stMsg.sText                                    := concat(_stMsg.sText, _ItfProcessCollector[E_INSTANCE.OUTFEED_ROBOT_R2].BitsToString(_wDisable));
              f_MessageSet(_stMsg);
            END_IF
          END_IF
        ELSE
          _InstanceCtrl[E_INSTANCE.OUTFEED_ROBOT_R2].Cmd      := E_INSTANCE_CMD.ENABLE;
        END_IF
      END_CASE

      E_INSTANCE_STATE.ENABLED:
        CASE _InstanceState[E_INSTANCE.OUTFEED_ROBOT_R2].Progress
        OF
          E_PROGRESS.PROGRESS_OCCUPIED:
            _InstanceCtrl[E_INSTANCE.OUTFEED_ROBOT_R2].Cmd    := E_INSTANCE_CMD.PROCEED;
        END_CASE

      E_INSTANCE_STATE.WORKING:
        CASE _InstanceState[E_INSTANCE.OUTFEED_ROBOT_R2].Progress
        OF
          E_PROGRESS.PROGRESS_BUSY:
            _tonProcess [E_INSTANCE.OUTFEED_ROBOT_R2]
                                                  (IN         := FALSE, 
                                                   PT         := _tProcess[E_INSTANCE.OUTFEED_ROBOT_R2]);

            _InstanceCtrl[E_INSTANCE.OUTFEED_ROBOT_R2].Cmd    := E_INSTANCE_CMD.WORK;

    
          E_PROGRESS.PROGRESS_CHECK:
            _tonProcess [E_INSTANCE.OUTFEED_ROBOT_R2]
                                                  (IN         := TRUE, 
                                                   PT         := _tProcess[E_INSTANCE.OUTFEED_ROBOT_R2]);
    
            IF _tonProcess [E_INSTANCE.OUTFEED_ROBOT_R2].Q
            THEN
              _InstanceCtrl[E_INSTANCE.OUTFEED_ROBOT_R2].Cmd  := E_INSTANCE_CMD.FINISH;
            END_IF
        END_CASE

      E_INSTANCE_STATE.FINISH:
        CASE _InstanceState[E_INSTANCE.OUTFEED_ROBOT_R2].Progress
        OF
          E_PROGRESS.PROGRESS_BUSY:
            _InstanceCtrl[E_INSTANCE.OUTFEED_ROBOT_R2].Cmd    := E_INSTANCE_CMD.FINISH;

          E_PROGRESS.PROGRESS_DONE:
            _InstanceCtrl[E_INSTANCE.OUTFEED_ROBOT_R2].Cmd    := E_INSTANCE_CMD.DISABLE;
        END_CASE
      END_CASE

    //-------------------------------------------------------------------------
    // E_INSTANCE.SENDER_FAST
    //-------------------------------------------------------------------------
    CASE _InstanceState[E_INSTANCE.SENDER_FAST].State
    OF
      E_INSTANCE_STATE.DISABLED:
        CASE _InstanceState[E_INSTANCE.SENDER_FAST].Progress
        OF
          E_PROGRESS.PROGRESS_BUSY:
            IF NOT (_ItfProcessCollector[E_INSTANCE.OUTFEED_ROBOT_R1].QueueProcessCount < 12) OR 
               NOT (_ItfProcessCollector[E_INSTANCE.OUTFEED_ROBOT_R2].QueueProcessCount < 12)
            THEN
              _InstanceCtrl[E_INSTANCE.SENDER_FAST].Cmd       := E_INSTANCE_CMD.ENABLE;

            ELSIF (_ItfProcessCollector[E_INSTANCE.SENDER_FAST].QueueProcessCount > 0)
            THEN
              _InstanceCtrl[E_INSTANCE.SENDER_FAST].Cmd       := E_INSTANCE_CMD.ENABLE;
            ELSE
              _InstanceCtrl[E_INSTANCE.SENDER_FAST].Cmd       := E_INSTANCE_CMD.DISABLE;

              IF NOT (_ItfProcessCollector[E_INSTANCE.SENDER_FAST].GetBit(_wDisable, TO_BYTE(E_INSTANCE.SENDER_FAST-1)))
              THEN
                _wDisable                                     := _ItfProcessCollector[E_INSTANCE.SENDER_FAST].
                                                                 SetBit(_wDisable, TO_BYTE(E_INSTANCE.SENDER_FAST-1));
    
                IF (_MessageLevel > E_MessageType.eMessageError)
                THEN
                  _stMsg.eType                                := E_MessageType.eMessageInfo;
                  _stMsg.eSubdevice                           := e_Subdevice.Application_Finish;
                  _stMsg.iErrorNumber                         := 0;
                  _stMsg.sText                                := concat(TO_STRING(E_INSTANCE.SENDER_FAST), ': _wDisable ');
                  _stMsg.sText                                := concat(_stMsg.sText, _ItfProcessCollector[E_INSTANCE.SENDER_FAST].BitsToString(_wDisable));
                  f_MessageSet(_stMsg);
                END_IF
              END_IF
            END_IF
        END_CASE

      E_INSTANCE_STATE.FINISH:
        CASE _InstanceState[E_INSTANCE.SENDER_FAST].Progress
        OF
          E_PROGRESS.PROGRESS_BUSY:
            _InstanceCtrl[E_INSTANCE.SENDER_FAST].Cmd         := E_INSTANCE_CMD.FINISH;
        END_CASE
      END_CASE
END_CASE
//-----------------------------------------------------------------------------
//-----------------------------------------------------------------------------
CASE _eState
OF
  E_PROGRESS.PROGRESS_STILL_WORKING:
    _XtsTransportCtrl.Cmd                                 := E_XTS_TRANSPORT_CTRL.CMD_GROUP_STOP;
  
    IF (_XtsTransportState.State = E_XTS_TRANSPORT_STATE.TRANSPORT_GROUP_STOP + E_PROGRESS.PROGRESS_ERROR)
    THEN
      _eState                                             := E_PROGRESS.PROGRESS_ERROR;

      _stMsg.eType                  := E_MessageType.eMessageError;
      _stMsg.eSubdevice             := e_Subdevice.Application_Finish;
      _stMsg.iErrorNumber           := 0;
      _stMsg.sText                  := concat(TO_STRING(_eState), ': ');
      f_MessageSet(_stMsg);

  
    ELSIF (_XtsTransportState.State = E_XTS_TRANSPORT_STATE.TRANSPORT_GROUP_STOP + E_PROGRESS.PROGRESS_DONE)
    THEN
      _eState                                             := E_PROGRESS.PROGRESS_DONE;

      IF (_MessageLevel > E_MessageType.eMessageError)
      THEN
        _stMsg.eType                := E_MessageType.eMessageInfo;
        _stMsg.eSubdevice           := e_Subdevice.Application_Finish;
        _stMsg.iErrorNumber         := 0;
        _stMsg.sText                := concat(TO_STRING(_eState), ': ');
        f_MessageSet(_stMsg);
      END_IF
    END_IF
END_CASE
//-----------------------------------------------------------------------------
//-----------------------------------------------------------------------------

Finish                            := _eState;
END_METHOD

METHOD Init       : E_PROGRESS // used only for first cycle startup, 
                               // use method Clear during operations if you have to clean up the instances 
VAR_INPUT
  Execute         : BOOL;
END_VAR
VAR_INST
  _nIdx,
  _nErrorId       : UDINT;
  _eState         : E_PROGRESS;
END_VAR
//-----------------------------------------------------------------------------
IF NOT Execute 
THEN 
	_eState                                         := E_PROGRESS.PROGRESS_INIT; 
END_IF 
//-----------------------------------------------------------------------------
IF NOT Check() 
THEN 
	Init                                            := E_PROGRESS.PROGRESS_ERROR; 
	RETURN; 
END_IF
//-----------------------------------------------------------------------------
//-----------------------------------------------------------------------------
CASE _eState
OF
  //---------------------------------------------------------------------------------------------------------------
  //---------------------------------------------------------------------------------------------------------------
  E_PROGRESS.PROGRESS_INIT:                   // startup procedure for your application
    IF Execute
    THEN
      _eState                                       := E_PROGRESS.PROGRESS_BUSY;

      IF (_MessageLevel > E_MessageType.eMessageError)
      THEN
        _stMsg.eType            := E_MessageType.eMessageInfo;
        _stMsg.eSubdevice       := e_Subdevice.Application_Init;
        _stMsg.iErrorNumber     := 0;
        _stMsg.sText            := concat(TO_STRING(_eState), ': ');
        f_MessageSet(_stMsg);
      END_IF
  
      FOR _nIdx := 1 TO MAX_PROCESS
      DO
        _InstanceCtrl[_nIdx].Cmd                    := E_INSTANCE_CMD.INIT;
      END_FOR
    END_IF
  //---------------------------------------------------------------------------------------------------------------
  //---------------------------------------------------------------------------------------------------------------
  E_PROGRESS.PROGRESS_BUSY:
    _InstanceCtrl[E_INSTANCE.BUFFER_INFEED].Cmd   := E_INSTANCE_CMD.DISABLE;
    //-----------------------------------------------------------------------------------
    CASE _InstanceState[E_INSTANCE.BUFFER_INFEED].State
    OF
      E_INSTANCE_STATE.DISABLED:
        CASE _InstanceState[E_INSTANCE.BUFFER_INFEED].Progress
        OF
          E_PROGRESS.PROGRESS_BUSY:           // check for startup to be done
            _eState                               := E_PROGRESS.PROGRESS_PREPARE; // go check next insatnce
        END_CASE
    END_CASE

  //---------------------------------------------------------------------------------------------------------------
  //---------------------------------------------------------------------------------------------------------------
  E_PROGRESS.PROGRESS_PREPARE:
    _InstanceCtrl[E_INSTANCE.INFEED].Cmd          := E_INSTANCE_CMD.DISABLE;
    //-----------------------------------------------------------------------------------
    CASE _InstanceState[E_INSTANCE.INFEED].State
    OF
      E_INSTANCE_STATE.DISABLED:
        CASE _InstanceState[E_INSTANCE.INFEED].Progress
        OF
          E_PROGRESS.PROGRESS_BUSY:           // check for startup to be done
          _eState                                 := E_PROGRESS.PROGRESS_STARTUP; // go check next insatnce
        END_CASE
    END_CASE

